C09128=1229.278,90.724,-47.007,-178.525,5.501,148.518
C09129=1229.283,90.475,-46.989,-178.527,5.501,148.519
C09130=1229.288,90.225,-46.971,-178.530,5.500,148.520
C09131=1229.292,89.976,-46.952,-178.532,5.499,148.520
C09132=1229.298,89.727,-46.933,-178.535,5.499,148.521
C09133=1229.303,89.478,-46.915,-178.537,5.498,148.521
C09134=1229.307,89.228,-46.898,-178.540,5.497,148.522
C09135=1229.312,88.979,-46.879,-178.542,5.496,148.522
C09136=1229.316,88.730,-46.860,-178.544,5.496,148.523
C09137=1229.321,88.481,-46.842,-178.548,5.494,148.524
C09138=1229.327,88.231,-46.824,-178.550,5.494,148.524
C09139=1229.331,87.981,-46.806,-178.552,5.493,148.525
C09140=1229.336,87.732,-46.788,-178.555,5.492,148.525
C09141=1229.341,87.483,-46.770,-178.558,5.492,148.526
C09142=1229.346,87.234,-46.752,-178.560,5.491,148.527
C09143=1229.351,86.985,-46.734,-178.562,5.490,148.527
C09144=1229.355,86.735,-46.715,-178.565,5.489,148.528
C09145=1229.360,86.486,-46.697,-178.568,5.489,148.528
C09146=1229.365,86.237,-46.678,-178.570,5.488,148.529
C09147=1229.370,85.988,-46.660,-178.572,5.487,148.529
C09148=1229.375,85.738,-46.642,-178.576,5.486,148.530
C09149=1229.380,85.489,-46.624,-178.578,5.485,148.531
C09150=1229.384,85.239,-46.606,-178.581,5.485,148.531
C09151=1229.389,84.990,-46.588,-178.583,5.484,148.532
C09152=1229.394,84.741,-46.570,-178.586,5.483,148.533
C09153=1229.399,84.492,-46.552,-178.588,5.482,148.533
C09154=1229.404,84.243,-46.534,-178.591,5.482,148.534
C09155=1229.408,83.993,-46.515,-178.593,5.481,148.534
C09156=1229.413,83.744,-46.497,-178.596,5.480,148.535
C09157=1229.418,83.494,-46.480,-178.598,5.480,148.536
C09158=1229.423,83.245,-46.462,-178.601,5.479,148.536
C09159=1229.428,82.996,-46.444,-178.604,5.479,148.537
C09160=1229.433,82.747,-46.426,-178.606,5.478,148.537
C09161=1229.438,82.498,-46.408,-178.609,5.476,148.538
C09162=1229.442,82.248,-46.389,-178.611,5.476,148.539
C09163=1229.448,81.979,-46.369,-178.614,5.475,148.539
C09164=1229.453,81.711,-46.350,-178.617,5.474,148.540
C09165=1229.459,81.443,-46.332,-178.619,5.474,148.541
C09166=1229.464,81.175,-46.312,-178.622,5.473,148.541
C09167=1229.468,80.925,-46.294,-178.625,5.472,148.542
C09168=1229.473,80.676,-46.276,-178.627,5.471,148.542
C09169=1229.478,80.426,-46.258,-178.630,5.470,148.543
C09170=1229.483,80.177,-46.240,-178.633,5.470,148.544
C09171=1229.488,79.928,-46.222,-178.635,5.469,148.544
C09172=1229.493,79.678,-46.205,-178.637,5.468,148.545
C09173=1229.498,79.429,-46.187,-178.640,5.467,148.545
C09174=1229.503,79.180,-46.169,-178.643,5.467,148.546
C09175=1229.508,78.931,-46.151,-178.645,5.466,148.547
C09176=1229.512,78.682,-46.133,-178.648,5.466,148.547
C09177=1229.517,78.433,-46.115,-178.650,5.465,148.548
C09178=1229.522,78.183,-46.098,-178.653,5.464,148.548
C09179=1229.527,77.933,-46.080,-178.655,5.464,148.549
C09180=1229.532,77.684,-46.062,-178.658,5.463,148.550
C09181=1229.537,77.435,-46.044,-178.660,5.462,148.550
C09182=1229.541,77.186,-46.026,-178.663,5.461,148.551
C09183=1229.547,76.936,-46.008,-178.665,5.461,148.551
C09184=1229.552,76.687,-45.990,-178.668,5.460,148.552
C09185=1229.556,76.438,-45.973,-178.670,5.460,148.553
C09186=1229.561,76.188,-45.955,-178.673,5.459,148.553
C09187=1229.566,75.939,-45.938,-178.676,5.457,148.554
C09188=1229.571,75.690,-45.920,-178.678,5.457,148.555
C09189=1229.576,75.440,-45.902,-178.681,5.456,148.555
C09190=1229.581,75.191,-45.885,-178.684,5.456,148.556
C09191=1229.586,74.941,-45.867,-178.686,5.455,148.556
C09192=1229.590,74.693,-45.849,-178.688,5.454,148.557
C09193=1229.595,74.443,-45.832,-178.691,5.453,148.558
C09194=1229.600,74.194,-45.814,-178.694,5.453,148.558
C09195=1229.605,73.944,-45.796,-178.696,5.452,148.559
C09196=1229.610,73.695,-45.779,-178.698,5.451,148.559
C09197=1229.614,73.446,-45.761,-178.701,5.451,148.560
C09198=1229.619,73.197,-45.743,-178.704,5.450,148.561
C09199=1229.625,72.947,-45.726,-178.706,5.449,148.561
C09200=1229.629,72.698,-45.708,-178.709,5.449,148.562
C09201=1229.634,72.448,-45.690,-178.711,5.448,148.562
C09202=1229.639,72.199,-45.674,-178.714,5.447,148.563
C09203=1229.644,71.950,-45.656,-178.716,5.447,148.564
C09204=1229.649,71.700,-45.638,-178.719,5.446,148.564
C09205=1229.654,71.451,-45.620,-178.722,5.446,148.565
C09206=1229.658,71.201,-45.604,-178.724,5.445,148.565
C09207=1229.663,70.952,-45.586,-178.726,5.444,148.566
C09208=1229.668,70.703,-45.568,-178.729,5.443,148.567
C09209=1229.673,70.453,-45.550,-178.732,5.443,148.567
C09210=1229.678,70.204,-45.533,-178.734,5.442,148.568
C09211=1229.683,69.954,-45.516,-178.737,5.442,148.569
C09212=1229.688,69.706,-45.498,-178.739,5.441,148.569
C09213=1229.693,69.457,-45.481,-178.742,5.440,148.570
C09214=1229.698,69.207,-45.463,-178.744,5.440,148.571
C09215=1229.703,68.958,-45.446,-178.747,5.439,148.571
C09216=1229.708,68.708,-45.428,-178.750,5.438,148.572
C09217=1229.712,68.459,-45.412,-178.752,5.438,148.572
C09218=1229.717,68.210,-45.394,-178.754,5.437,148.573
C09219=1229.722,67.960,-45.376,-178.757,5.436,148.574
C09220=1229.727,67.710,-45.360,-178.760,5.436,148.574
C09221=1229.732,67.461,-45.342,-178.762,5.435,148.575
C09222=1229.736,67.212,-45.325,-178.765,5.435,148.576
C09223=1229.741,66.963,-45.307,-178.767,5.434,148.576
C09224=1229.747,66.713,-45.290,-178.770,5.433,148.577
C09225=1229.751,66.465,-45.273,-178.772,5.432,148.577
C09226=1229.756,66.215,-45.255,-178.775,5.432,148.578
C09227=1229.762,65.965,-45.238,-178.777,5.431,148.579
C09228=1229.766,65.716,-45.221,-178.780,5.431,148.579
C09229=1229.771,65.466,-45.204,-178.782,5.430,148.580
C09230=1229.776,65.217,-45.187,-178.785,5.429,148.580
C09231=1229.780,64.968,-45.169,-178.788,5.429,148.581
C09232=1229.786,64.719,-45.152,-178.790,5.428,148.582
C09233=1229.791,64.469,-45.135,-178.793,5.427,148.582
C09234=1229.796,64.220,-45.117,-178.795,5.427,148.583
C09235=1229.800,63.970,-45.101,-178.798,5.426,148.584
C09236=1229.805,63.721,-45.083,-178.800,5.425,148.584
C09237=1229.810,63.471,-45.065,-178.803,5.425,148.585
C09238=1229.815,63.222,-45.049,-178.805,5.424,148.586
C09239=1229.821,62.973,-45.032,-178.808,5.424,148.586
C09240=1229.825,62.724,-45.015,-178.811,5.423,148.587
C09241=1229.830,62.474,-44.997,-178.813,5.422,148.588
C09242=1229.834,62.225,-44.981,-178.815,5.421,148.588
C09243=1229.840,61.975,-44.963,-178.818,5.421,148.589
C09244=1229.844,61.726,-44.946,-178.821,5.420,148.589
C09245=1229.850,61.477,-44.929,-178.823,5.420,148.590
C09246=1229.854,61.228,-44.912,-178.825,5.420,148.591
C09247=1229.859,60.978,-44.895,-178.828,5.419,148.591
C09248=1229.864,60.728,-44.878,-178.831,5.419,148.592
C09249=1229.869,60.479,-44.860,-178.833,5.418,148.592
C09250=1229.874,60.230,-44.844,-178.835,5.417,148.593
C09251=1229.879,59.981,-44.827,-178.838,5.417,148.594
C09252=1229.884,59.731,-44.810,-178.841,5.416,148.594
C09253=1229.889,59.481,-44.793,-178.843,5.416,148.595
C09254=1229.894,59.232,-44.777,-178.846,5.415,148.596
C09255=1229.899,58.983,-44.759,-178.849,5.414,148.596
C09256=1229.903,58.734,-44.742,-178.851,5.413,148.597
C09257=1229.908,58.484,-44.725,-178.853,5.413,148.597
C09258=1229.913,58.234,-44.708,-178.856,5.412,148.598
C09259=1229.918,57.986,-44.692,-178.859,5.412,148.599
C09260=1229.923,57.736,-44.674,-178.861,5.411,148.599
C09261=1229.928,57.486,-44.658,-178.864,5.411,148.600
C09262=1229.933,57.237,-44.641,-178.867,5.410,148.601
C09263=1229.938,56.988,-44.624,-178.869,5.409,148.601
C09264=1229.943,56.739,-44.606,-178.871,5.409,148.602
C09265=1229.947,56.489,-44.590,-178.874,5.408,148.603
C09266=1229.952,56.240,-44.573,-178.877,5.407,148.603
C09267=1229.958,55.972,-44.555,-178.879,5.407,148.604
C09268=1229.963,55.703,-44.538,-178.882,5.406,148.605
C09269=1229.969,55.434,-44.519,-178.885,5.406,148.605
C09270=1229.973,55.166,-44.501,-178.887,5.405,148.606
C09271=1229.979,54.917,-44.484,-178.890,5.404,148.607
C09272=1229.984,54.667,-44.467,-178.892,5.404,148.607
C09273=1229.988,54.418,-44.451,-178.895,5.403,148.608
C09274=1229.994,54.168,-44.434,-178.898,5.403,148.609
C09275=1229.999,53.919,-44.417,-178.900,5.402,148.609
C09276=1230.003,53.670,-44.400,-178.902,5.402,148.610
C09277=1230.008,53.421,-44.384,-178.905,5.402,148.611
C09278=1230.013,53.171,-44.367,-178.907,5.401,148.611
C09279=1230.018,52.921,-44.350,-178.910,5.400,148.612
C09280=1230.023,52.673,-44.334,-178.912,5.400,148.612
C09281=1230.028,52.423,-44.317,-178.915,5.399,148.613
C09282=1230.033,52.173,-44.300,-178.918,5.399,148.614
C09283=1230.037,51.924,-44.283,-178.920,5.398,148.614
C09284=1230.043,51.675,-44.266,-178.923,5.397,148.615
C09285=1230.047,51.425,-44.250,-178.926,5.397,148.616
C09286=1230.053,51.176,-44.234,-178.928,5.396,148.616
C09287=1230.057,50.926,-44.217,-178.930,5.395,148.617
C09288=1230.062,50.677,-44.200,-178.933,5.395,148.618
C09289=1230.068,50.428,-44.184,-178.935,5.395,148.618
C09290=1230.072,50.178,-44.167,-178.938,5.395,148.619
C09291=1230.076,49.929,-44.150,-178.940,5.394,148.620
C09292=1230.082,49.680,-44.134,-178.943,5.393,148.620
C09293=1230.087,49.430,-44.118,-178.946,5.393,148.621
C09294=1230.092,49.180,-44.101,-178.948,5.392,148.622
C09295=1230.097,48.931,-44.085,-178.951,5.392,148.622
C09296=1230.102,48.682,-44.067,-178.953,5.391,148.623
C09297=1230.107,48.433,-44.051,-178.956,5.390,148.623
C09298=1230.112,48.183,-44.035,-178.958,5.390,148.624
C09299=1230.116,47.933,-44.018,-178.961,5.389,148.625
C09300=1230.121,47.684,-44.002,-178.963,5.389,148.625
C09301=1230.127,47.435,-43.985,-178.966,5.389,148.626
C09302=1230.131,47.185,-43.968,-178.968,5.388,148.627
C09303=1230.136,46.936,-43.953,-178.971,5.388,148.627
C09304=1230.141,46.686,-43.936,-178.974,5.387,148.628
C09305=1230.146,46.438,-43.920,-178.976,5.386,148.629
C09306=1230.151,46.187,-43.904,-178.978,5.386,148.629
C09307=1230.157,45.938,-43.887,-178.981,5.385,148.630
C09308=1230.161,45.689,-43.870,-178.984,5.384,148.630
C09309=1230.166,45.439,-43.853,-178.986,5.384,148.631
C09310=1230.171,45.190,-43.838,-178.988,5.384,148.632
C09311=1230.175,44.940,-43.821,-178.991,5.384,148.632
C09312=1230.180,44.692,-43.805,-178.994,5.383,148.633
C09313=1230.185,44.442,-43.789,-178.996,5.382,148.634
C09314=1230.190,44.193,-43.773,-178.999,5.382,148.635
C09315=1230.196,43.943,-43.755,-179.002,5.381,148.635
C09316=1230.201,43.694,-43.740,-179.004,5.381,148.636
C09317=1230.205,43.444,-43.723,-179.006,5.380,148.636
C09318=1230.210,43.194,-43.707,-179.009,5.379,148.637
C09319=1230.215,42.945,-43.691,-179.011,5.379,148.638
C09320=1230.220,42.696,-43.674,-179.014,5.379,148.638
C09321=1230.225,42.446,-43.659,-179.016,5.378,148.639
C09322=1230.230,42.197,-43.642,-179.019,5.378,148.640
C09323=1230.235,41.947,-43.626,-179.022,5.377,148.640
C09324=1230.239,41.698,-43.610,-179.024,5.377,148.641
C09325=1230.245,41.449,-43.593,-179.027,5.376,148.642
C09326=1230.249,41.199,-43.577,-179.030,5.376,148.642
C09327=1230.254,40.950,-43.561,-179.032,5.376,148.643
C09328=1230.259,40.700,-43.545,-179.034,5.375,148.644
C09329=1230.264,40.451,-43.529,-179.036,5.374,148.644
C09330=1230.269,40.201,-43.513,-179.039,5.374,148.645
C09331=1230.275,39.952,-43.496,-179.042,5.373,148.646
C09332=1230.280,39.702,-43.480,-179.044,5.373,148.646
C09333=1230.285,39.453,-43.464,-179.047,5.372,148.647
C09334=1230.290,39.203,-43.448,-179.050,5.371,148.648
C09335=1230.295,38.954,-43.431,-179.052,5.372,148.648
C09336=1230.300,38.705,-43.416,-179.054,5.371,148.649
C09337=1230.305,38.456,-43.399,-179.057,5.371,148.650
C09338=1230.309,38.206,-43.384,-179.060,5.370,148.650
C09339=1230.314,37.957,-43.368,-179.062,5.369,148.651
C09340=1230.319,37.708,-43.352,-179.065,5.369,148.652
C09341=1230.324,37.457,-43.336,-179.068,5.368,148.652
C09342=1230.329,37.209,-43.320,-179.070,5.369,148.653
C09343=1230.334,36.959,-43.304,-179.072,5.368,148.653
C09344=1230.339,36.710,-43.287,-179.074,5.367,148.654
C09345=1230.344,36.460,-43.271,-179.077,5.367,148.655
C09346=1230.349,36.211,-43.255,-179.080,5.366,148.655
C09347=1230.354,35.962,-43.240,-179.082,5.365,148.656
C09348=1230.359,35.711,-43.224,-179.085,5.365,148.657
C09349=1230.364,35.463,-43.207,-179.087,5.365,148.657
C09350=1230.369,35.213,-43.191,-179.090,5.365,148.658
C09351=1230.374,34.963,-43.176,-179.092,5.364,148.659
C09352=1230.379,34.714,-43.160,-179.095,5.363,148.659
C09353=1230.383,34.465,-43.144,-179.098,5.363,148.660
C09354=1230.389,34.215,-43.129,-179.100,5.362,148.661
C09355=1230.393,33.966,-43.112,-179.102,5.363,148.662
C09356=1230.398,33.716,-43.096,-179.105,5.362,148.662
C09357=1230.404,33.467,-43.081,-179.108,5.362,148.663
C09358=1230.408,33.217,-43.064,-179.110,5.361,148.664
C09359=1230.414,32.968,-43.048,-179.112,5.360,148.664
C09360=1230.418,32.718,-43.033,-179.115,5.359,148.665
C09361=1230.423,32.469,-43.017,-179.118,5.359,148.665
C09362=1230.428,32.220,-43.001,-179.120,5.359,148.666
C09363=1230.433,31.970,-42.985,-179.122,5.359,148.667
C09364=1230.438,31.721,-42.970,-179.125,5.358,148.667
C09365=1230.443,31.472,-42.953,-179.128,5.358,148.668
C09366=1230.448,31.222,-42.937,-179.130,5.357,148.669
C09367=1230.453,30.973,-42.922,-179.133,5.356,148.669
C09368=1230.458,30.722,-42.906,-179.135,5.357,148.670
C09369=1230.463,30.473,-42.891,-179.138,5.356,148.671
C09370=1230.468,30.224,-42.875,-179.140,5.356,148.671
C09371=1230.474,29.956,-42.858,-179.143,5.355,148.672
C09372=1230.478,29.686,-42.841,-179.146,5.354,148.673
C09373=1230.484,29.418,-42.824,-179.148,5.354,148.673
C09374=1230.489,29.149,-42.807,-179.151,5.354,148.674
C09375=1230.495,28.900,-42.792,-179.154,5.353,148.675
C09376=1230.499,28.650,-42.775,-179.157,5.353,148.676
C09377=1230.504,28.401,-42.760,-179.158,5.353,148.676
C09378=1230.509,28.152,-42.745,-179.161,5.352,148.677
C09379=1230.514,27.902,-42.729,-179.164,5.351,148.678
C09380=1230.519,27.652,-42.713,-179.166,5.351,148.678
C09381=1230.524,27.403,-42.698,-179.169,5.350,148.679
C09382=1230.529,27.154,-42.682,-179.171,5.351,148.680
C09383=1230.534,26.904,-42.667,-179.174,5.350,148.680
C09384=1230.539,26.655,-42.652,-179.176,5.349,148.681
C09385=1230.544,26.406,-42.635,-179.179,5.349,148.682
C09386=1230.549,26.156,-42.619,-179.181,5.348,148.682
C09387=1230.554,25.906,-42.604,-179.184,5.348,148.683
C09388=1230.559,25.657,-42.589,-179.186,5.348,148.684
C09389=1230.564,25.408,-42.573,-179.189,5.348,148.684
C09390=1230.569,25.158,-42.557,-179.191,5.347,148.685
C09391=1230.574,24.909,-42.542,-179.194,5.346,148.686
C09392=1230.579,24.659,-42.527,-179.197,5.346,148.686
C09393=1230.584,24.410,-42.511,-179.199,5.346,148.687
C09394=1230.588,24.160,-42.496,-179.201,5.346,148.688
C09395=1230.594,23.911,-42.480,-179.204,5.345,148.688
C09396=1230.599,23.661,-42.464,-179.207,5.345,148.689
C09397=1230.604,23.412,-42.449,-179.209,5.344,148.690
C09398=1230.609,23.162,-42.434,-179.211,5.344,148.690
C09399=1230.613,22.913,-42.419,-179.214,5.344,148.691
C09400=1230.619,22.664,-42.403,-179.217,5.343,148.692
C09401=1230.624,22.414,-42.387,-179.219,5.343,148.693
C09402=1230.628,22.164,-42.372,-179.222,5.342,148.693
C09403=1230.634,21.915,-42.356,-179.224,5.342,148.694
C09404=1230.638,21.665,-42.342,-179.227,5.342,148.695
C09405=1230.644,21.416,-42.327,-179.229,5.341,148.695
C09406=1230.649,21.167,-42.311,-179.232,5.341,148.696
C09407=1230.653,20.917,-42.296,-179.234,5.340,148.696
C09408=1230.659,20.667,-42.280,-179.236,5.340,148.697
C09409=1230.663,20.418,-42.265,-179.239,5.339,148.698
C09410=1230.669,20.169,-42.249,-179.242,5.339,148.698
C09411=1230.674,19.919,-42.234,-179.244,5.338,148.699
C09412=1230.678,19.670,-42.218,-179.247,5.338,148.700
C09413=1230.684,19.420,-42.204,-179.249,5.338,148.700
C09414=1230.688,19.171,-42.189,-179.252,5.338,148.701
C09415=1230.694,18.921,-42.173,-179.254,5.337,148.702
C09416=1230.699,18.672,-42.158,-179.257,5.336,148.703
C09417=1230.703,18.422,-42.142,-179.259,5.337,148.703
C09418=1230.708,18.173,-42.127,-179.262,5.336,148.704
C09419=1230.714,17.923,-42.112,-179.264,5.336,148.705
C09420=1230.718,17.674,-42.097,-179.267,5.335,148.705
C09421=1230.724,17.424,-42.082,-179.270,5.335,148.706
C09422=1230.728,17.175,-42.067,-179.272,5.335,148.707
C09423=1230.733,16.925,-42.051,-179.274,5.334,148.707
C09424=1230.738,16.675,-42.036,-179.277,5.334,148.708
C09425=1230.743,16.426,-42.021,-179.280,5.333,148.709
C09426=1230.748,16.177,-42.006,-179.282,5.334,148.709
C09427=1230.753,15.928,-41.990,-179.284,5.333,148.710
C09428=1230.758,15.678,-41.976,-179.287,5.332,148.711
C09429=1230.764,15.428,-41.960,-179.290,5.332,148.711
C09430=1230.768,15.179,-41.945,-179.292,5.331,148.712
C09431=1230.773,14.929,-41.929,-179.294,5.332,148.713
C09432=1230.778,14.680,-41.915,-179.297,5.331,148.713
C09433=1230.784,14.430,-41.900,-179.300,5.331,148.714
C09434=1230.788,14.181,-41.885,-179.302,5.330,148.715
C09435=1230.793,13.931,-41.870,-179.304,5.330,148.716
C09436=1230.799,13.682,-41.855,-179.307,5.330,148.716
C09437=1230.803,13.433,-41.840,-179.310,5.329,148.717
C09438=1230.809,13.183,-41.825,-179.312,5.329,148.718
C09439=1230.814,12.934,-41.810,-179.314,5.329,148.718
C09440=1230.818,12.684,-41.794,-179.317,5.328,148.719
C09441=1230.823,12.434,-41.780,-179.320,5.328,148.720
C09442=1230.828,12.185,-41.765,-179.322,5.327,148.720
C09443=1230.834,11.935,-41.750,-179.324,5.328,148.721
C09444=1230.838,11.686,-41.735,-179.327,5.327,148.722
C09445=1230.843,11.437,-41.720,-179.330,5.327,148.722
C09446=1230.849,11.187,-41.705,-179.332,5.326,148.723
C09447=1230.853,10.938,-41.690,-179.334,5.326,148.724
C09448=1230.858,10.688,-41.676,-179.337,5.326,148.724
C09449=1230.864,10.438,-41.660,-179.340,5.325,148.725
C09450=1230.868,10.189,-41.645,-179.342,5.325,148.726
C09451=1230.873,9.940,-41.631,-179.344,5.325,148.726
C09452=1230.879,9.690,-41.615,-179.347,5.324,148.727
C09453=1230.884,9.440,-41.601,-179.350,5.324,148.728
C09454=1230.888,9.191,-41.586,-179.352,5.323,148.729
C09455=1230.894,8.941,-41.571,-179.354,5.324,148.729
C09456=1230.899,8.692,-41.556,-179.357,5.323,148.730
C09457=1230.904,8.443,-41.542,-179.360,5.323,148.731
C09458=1230.909,8.193,-41.526,-179.362,5.322,148.731
C09459=1230.914,7.943,-41.512,-179.365,5.322,148.732
C09460=1230.918,7.694,-41.497,-179.367,5.322,148.733
C09461=1230.924,7.444,-41.482,-179.370,5.321,148.733
C09462=1230.928,7.195,-41.467,-179.372,5.321,148.734
C09463=1230.933,6.945,-41.452,-179.375,5.321,148.735
C09464=1230.938,6.696,-41.437,-179.377,5.320,148.735
C09465=1230.944,6.446,-41.423,-179.380,5.320,148.736
C09466=1230.948,6.197,-41.408,-179.382,5.319,148.737
C09467=1230.953,5.947,-41.393,-179.385,5.320,148.737
C09468=1230.958,5.697,-41.379,-179.387,5.319,148.738
C09469=1230.964,5.448,-41.363,-179.390,5.319,148.739
C09470=1230.969,5.199,-41.349,-179.393,5.318,148.740
C09471=1230.974,4.950,-41.334,-179.395,5.318,148.740
C09472=1230.979,4.700,-41.320,-179.397,5.318,148.741
C09473=1230.984,4.450,-41.305,-179.400,5.317,148.742
C09474=1230.989,4.201,-41.290,-179.402,5.318,148.742
C09475=1230.994,3.932,-41.275,-179.405,5.317,148.743
C09476=1230.999,3.663,-41.259,-179.408,5.317,148.744
C09477=1231.005,3.394,-41.243,-179.410,5.316,148.745
C09478=1231.011,3.125,-41.228,-179.413,5.316,148.745
C09479=1231.015,2.876,-41.213,-179.416,5.315,148.746
C09480=1231.020,2.626,-41.198,-179.418,5.316,148.747
C09481=1231.025,2.376,-41.184,-179.420,5.315,148.747
C09482=1231.031,2.127,-41.169,-179.423,5.314,148.748
C09483=1231.035,1.877,-41.154,-179.426,5.314,148.749
C09484=1231.040,1.627,-41.140,-179.428,5.314,148.749
C09485=1231.045,1.378,-41.125,-179.431,5.314,148.750
C09486=1231.050,1.129,-41.111,-179.433,5.313,148.751
C09487=1231.056,0.880,-41.097,-179.435,5.313,148.751
C09488=1231.061,0.630,-41.082,-179.438,5.313,148.752
C09489=1231.066,0.381,-41.067,-179.441,5.312,148.753
C09490=1231.071,0.131,-41.053,-179.443,5.312,148.754
C09491=1231.076,-0.119,-41.038,-179.445,5.312,148.754
C09492=1231.081,-0.369,-41.024,-179.448,5.312,148.755
C09493=1231.085,-0.618,-41.009,-179.451,5.311,148.756
C09494=1231.090,-0.867,-40.995,-179.453,5.311,148.756
C09495=1231.095,-1.117,-40.981,-179.455,5.311,148.757
C09496=1231.100,-1.367,-40.966,-179.458,5.310,148.758
C09497=1231.106,-1.616,-40.952,-179.461,5.310,148.758
C09498=1231.111,-1.865,-40.937,-179.463,5.310,148.759
C09499=1231.116,-2.115,-40.922,-179.465,5.310,148.760
C09500=1231.121,-2.365,-40.908,-179.468,5.309,148.760
C09501=1231.126,-2.614,-40.894,-179.470,5.309,148.761
C09502=1231.131,-2.864,-40.880,-179.473,5.309,148.762
C09503=1231.136,-3.114,-40.865,-179.475,5.308,148.762
C09504=1231.141,-3.363,-40.850,-179.477,5.309,148.763
C09505=1231.146,-3.612,-40.836,-179.480,5.308,148.764
C09506=1231.151,-3.862,-40.822,-179.483,5.307,148.765
C09507=1231.156,-4.111,-40.808,-179.486,5.307,148.765
C09508=1231.161,-4.361,-40.794,-179.488,5.308,148.766
C09509=1231.166,-4.611,-40.779,-179.491,5.307,148.767
C09510=1231.171,-4.860,-40.765,-179.493,5.307,148.768
C09511=1231.177,-5.109,-40.751,-179.495,5.307,148.768
C09512=1231.182,-5.359,-40.737,-179.498,5.306,148.769
C09513=1231.186,-5.608,-40.722,-179.501,5.306,148.770
C09514=1231.191,-5.858,-40.708,-179.503,5.306,148.770
C09515=1231.196,-6.108,-40.693,-179.505,5.306,148.771
C09516=1231.201,-6.357,-40.679,-179.508,5.305,148.772
C09517=1231.207,-6.606,-40.665,-179.511,5.305,148.772
C09518=1231.212,-6.856,-40.651,-179.513,5.305,148.773
C09519=1231.216,-7.106,-40.637,-179.515,5.304,148.774
C09520=1231.221,-7.356,-40.622,-179.518,5.304,148.774
C09521=1231.226,-7.605,-40.608,-179.520,5.304,148.775
C09522=1231.232,-7.854,-40.594,-179.523,5.304,148.776
C09523=1231.237,-8.104,-40.580,-179.526,5.303,148.777
C09524=1231.242,-8.354,-40.566,-179.528,5.303,148.777
C09525=1231.247,-8.603,-40.551,-179.530,5.303,148.778
C09526=1231.252,-8.853,-40.537,-179.533,5.302,148.779
C09527=1231.257,-9.102,-40.524,-179.535,5.303,148.779
C09528=1231.262,-9.352,-40.509,-179.538,5.302,148.780
C09529=1231.266,-9.601,-40.495,-179.540,5.302,148.781
C09530=1231.271,-9.851,-40.481,-179.542,5.302,148.781
C09531=1231.277,-10.100,-40.467,-179.545,5.301,148.782
C09532=1231.282,-10.350,-40.453,-179.548,5.301,148.783
C09533=1231.287,-10.600,-40.439,-179.550,5.300,148.783
C09534=1231.292,-10.850,-40.425,-179.552,5.301,148.784
C09535=1231.298,-11.099,-40.411,-179.555,5.300,148.785
C09536=1231.303,-11.348,-40.397,-179.558,5.300,148.786
C09537=1231.307,-11.598,-40.383,-179.560,5.300,148.786
C09538=1231.312,-11.848,-40.369,-179.562,5.299,148.787
C09539=1231.317,-12.097,-40.355,-179.565,5.299,148.788
C09540=1231.322,-12.346,-40.341,-179.567,5.299,148.788
C09541=1231.327,-12.596,-40.326,-179.570,5.299,148.789
C09542=1231.333,-12.846,-40.313,-179.573,5.298,148.790
C09543=1231.337,-13.095,-40.299,-179.575,5.299,148.791
C09544=1231.342,-13.345,-40.285,-179.578,5.298,148.791
C09545=1231.347,-13.594,-40.271,-179.580,5.298,148.792
C09546=1231.353,-13.843,-40.257,-179.582,5.298,148.793
C09547=1231.358,-14.093,-40.243,-179.585,5.297,148.793
C09548=1231.363,-14.343,-40.229,-179.588,5.297,148.794
C09549=1231.368,-14.592,-40.216,-179.590,5.297,148.795
C09550=1231.373,-14.842,-40.201,-179.593,5.297,148.795
C09551=1231.378,-15.092,-40.187,-179.595,5.296,148.796
C09552=1231.383,-15.341,-40.173,-179.597,5.296,148.797
C09553=1231.389,-15.591,-40.160,-179.600,5.296,148.798
C09554=1231.393,-15.840,-40.146,-179.603,5.295,148.798
C09555=1231.398,-16.090,-40.132,-179.605,5.296,148.799
C09556=1231.403,-16.339,-40.118,-179.607,5.295,148.800
C09557=1231.409,-16.589,-40.104,-179.610,5.295,148.800
C09558=1231.413,-16.839,-40.091,-179.612,5.295,148.801
C09559=1231.418,-17.088,-40.077,-179.615,5.295,148.802
C09560=1231.423,-17.337,-40.062,-179.617,5.294,148.802
C09561=1231.429,-17.588,-40.049,-179.619,5.294,148.803
C09562=1231.433,-17.837,-40.036,-179.622,5.294,148.804
C09563=1231.438,-18.086,-40.021,-179.625,5.293,148.804
C09564=1231.444,-18.337,-40.008,-179.627,5.294,148.805
C09565=1231.449,-18.586,-39.994,-179.630,5.293,148.806
C09566=1231.453,-18.835,-39.980,-179.632,5.293,148.807
C09567=1231.459,-19.085,-39.967,-179.634,5.293,148.807
C09568=1231.464,-19.334,-39.953,-179.637,5.292,148.808
C09569=1231.468,-19.584,-39.939,-179.639,5.293,148.809
C09570=1231.474,-19.833,-39.926,-179.642,5.292,148.810
C09571=1231.479,-20.083,-39.911,-179.645,5.292,148.810
C09572=1231.484,-20.333,-39.897,-179.647,5.292,148.811
C09573=1231.489,-20.582,-39.885,-179.650,5.292,148.812
C09574=1231.494,-20.832,-39.870,-179.652,5.291,148.812
C09575=1231.500,-21.081,-39.857,-179.654,5.292,148.813
C09576=1231.504,-21.331,-39.843,-179.657,5.291,148.814
C09577=1231.509,-21.581,-39.829,-179.660,5.291,148.814
C09578=1231.515,-21.830,-39.816,-179.662,5.291,148.815
C09579=1231.520,-22.099,-39.802,-179.664,5.290,148.816
C09580=1231.525,-22.369,-39.787,-179.667,5.290,148.817
C09581=1231.531,-22.637,-39.772,-179.670,5.290,148.817
C09582=1231.537,-22.907,-39.757,-179.672,5.290,148.818
C09583=1231.541,-23.157,-39.744,-179.675,5.289,148.819
C09584=1231.547,-23.406,-39.730,-179.678,5.289,148.820
C09585=1231.552,-23.656,-39.717,-179.680,5.289,148.820
C09586=1231.557,-23.905,-39.703,-179.682,5.289,148.821
C09587=1231.562,-24.155,-39.690,-179.685,5.288,148.822
C09588=1231.566,-24.405,-39.676,-179.687,5.289,148.822
C09589=1231.572,-24.654,-39.663,-179.690,5.288,148.823
C09590=1231.577,-24.904,-39.649,-179.692,5.288,148.824
C09591=1231.582,-25.153,-39.636,-179.694,5.288,148.824
C09592=1231.587,-25.403,-39.622,-179.697,5.287,148.825
C09593=1231.592,-25.652,-39.609,-179.699,5.288,148.826
C09594=1231.597,-25.902,-39.595,-179.702,5.287,148.827
C09595=1231.603,-26.151,-39.582,-179.705,5.287,148.827
C09596=1231.607,-26.401,-39.568,-179.707,5.287,148.828
C09597=1231.612,-26.651,-39.555,-179.710,5.287,148.829
C09598=1231.618,-26.901,-39.542,-179.712,5.287,148.830
C09599=1231.622,-27.150,-39.528,-179.715,5.287,148.830
C09600=1231.628,-27.400,-39.515,-179.717,5.286,148.831
C09601=1231.633,-27.649,-39.501,-179.719,5.286,148.832
C09602=1231.638,-27.899,-39.488,-179.722,5.286,148.832
C09603=1231.643,-28.149,-39.474,-179.725,5.285,148.833
C09604=1231.648,-28.398,-39.461,-179.727,5.286,148.834
C09605=1231.653,-28.648,-39.447,-179.729,5.285,148.834
C09606=1231.658,-28.897,-39.434,-179.731,5.286,148.835
C09607=1231.663,-29.147,-39.421,-179.734,5.285,148.836
C09608=1231.669,-29.396,-39.408,-179.737,5.285,148.837
C09609=1231.674,-29.646,-39.394,-179.739,5.285,148.837
C09610=1231.679,-29.895,-39.381,-179.741,5.284,148.838
C09611=1231.684,-30.146,-39.368,-179.744,5.284,148.839
C09612=1231.689,-30.394,-39.354,-179.746,5.284,148.839
C09613=1231.693,-30.644,-39.341,-179.749,5.284,148.840
C09614=1231.699,-30.894,-39.328,-179.751,5.284,148.841
C09615=1231.704,-31.143,-39.315,-179.754,5.283,148.841
C09616=1231.709,-31.393,-39.301,-179.756,5.283,148.842
C09617=1231.714,-31.642,-39.289,-179.758,5.283,148.843
C09618=1231.720,-31.893,-39.275,-179.762,5.283,148.844
C09619=1231.724,-32.141,-39.262,-179.764,5.283,148.844
C09620=1231.730,-32.392,-39.248,-179.766,5.283,148.845
C09621=1231.735,-32.641,-39.236,-179.769,5.282,148.846
C09622=1231.739,-32.891,-39.222,-179.771,5.283,148.847
C09623=1231.745,-33.140,-39.209,-179.774,5.282,148.847
C09624=1231.749,-33.390,-39.196,-179.776,5.282,148.848
C09625=1231.755,-33.640,-39.183,-179.778,5.282,148.849
C09626=1231.760,-33.889,-39.170,-179.781,5.282,148.849
C09627=1231.765,-34.139,-39.156,-179.783,5.282,148.850
C09628=1231.770,-34.388,-39.143,-179.786,5.281,148.851
C09629=1231.775,-34.638,-39.130,-179.788,5.281,148.851
C09630=1231.781,-34.888,-39.117,-179.791,5.281,148.852
C09631=1231.786,-35.137,-39.104,-179.793,5.281,148.853
C09632=1231.790,-35.387,-39.091,-179.795,5.281,148.854
C09633=1231.796,-35.636,-39.077,-179.798,5.280,148.854
C09634=1231.801,-35.886,-39.064,-179.801,5.280,148.855
C09635=1231.806,-36.135,-39.052,-179.803,5.280,148.856
C09636=1231.812,-36.385,-39.039,-179.805,5.280,148.856
C09637=1231.816,-36.635,-39.026,-179.807,5.280,148.857
C09638=1231.821,-36.884,-39.012,-179.810,5.280,148.858
C09639=1231.826,-37.134,-38.999,-179.813,5.279,148.859
C09640=1231.831,-37.383,-38.986,-179.815,5.280,148.859
C09641=1231.836,-37.633,-38.974,-179.818,5.279,148.860
C09642=1231.842,-37.883,-38.960,-179.820,5.280,148.861
C09643=1231.847,-38.132,-38.947,-179.823,5.279,148.861
C09644=1231.852,-38.382,-38.935,-179.825,5.279,148.862
C09645=1231.857,-38.632,-38.921,-179.828,5.279,148.863
C09646=1231.862,-38.881,-38.909,-179.830,5.278,148.864
C09647=1231.867,-39.131,-38.896,-179.832,5.279,148.864
C09648=1231.872,-39.380,-38.882,-179.835,5.278,148.865
C09649=1231.877,-39.630,-38.869,-179.838,5.278,148.866
C09650=1231.882,-39.880,-38.856,-179.840,5.278,148.866
C09651=1231.887,-40.129,-38.844,-179.842,5.278,148.867
C09652=1231.893,-40.379,-38.830,-179.844,5.278,148.868
C09653=1231.897,-40.629,-38.817,-179.847,5.277,148.868
C09654=1231.903,-40.878,-38.805,-179.850,5.277,148.869
C09655=1231.908,-41.127,-38.792,-179.852,5.277,148.870
C09656=1231.913,-41.378,-38.779,-179.855,5.277,148.871
C09657=1231.918,-41.627,-38.766,-179.857,5.277,148.871
C09658=1231.923,-41.876,-38.754,-179.859,5.277,148.872
C09659=1231.928,-42.126,-38.741,-179.861,5.277,148.873
C09660=1231.933,-42.376,-38.728,-179.864,5.276,148.873
C09661=1231.939,-42.625,-38.715,-179.867,5.276,148.874
C09662=1231.944,-42.875,-38.702,-179.869,5.277,148.875
C09663=1231.948,-43.125,-38.689,-179.872,5.276,148.876
C09664=1231.954,-43.374,-38.677,-179.874,5.276,148.876
C09665=1231.959,-43.623,-38.664,-179.877,5.276,148.877
C09666=1231.964,-43.874,-38.651,-179.879,5.275,148.878
C09667=1231.969,-44.124,-38.639,-179.881,5.276,148.878
C09668=1231.974,-44.373,-38.626,-179.884,5.275,148.879
C09669=1231.980,-44.622,-38.613,-179.886,5.276,148.880
C09670=1231.984,-44.872,-38.600,-179.889,5.275,148.881
C09671=1231.989,-45.122,-38.588,-179.891,5.275,148.881
C09672=1231.995,-45.371,-38.575,-179.894,5.275,148.882
C09673=1232.000,-45.621,-38.562,-179.896,5.274,148.883
C09674=1232.005,-45.870,-38.549,-179.898,5.275,148.883
C09675=1232.010,-46.120,-38.536,-179.901,5.274,148.884
C09676=1232.015,-46.370,-38.525,-179.903,5.275,148.885
C09677=1232.020,-46.620,-38.512,-179.906,5.274,148.886
C09678=1232.025,-46.869,-38.499,-179.908,5.274,148.886
C09679=1232.031,-47.119,-38.486,-179.910,5.274,148.887
C09680=1232.036,-47.368,-38.473,-179.913,5.273,148.888
C09681=1232.040,-47.618,-38.460,-179.915,5.274,148.888
C09682=1232.046,-47.868,-38.448,-179.918,5.273,148.889
C09683=1232.051,-48.137,-38.435,-179.920,5.274,148.890
C09684=1232.057,-48.407,-38.421,-179.923,5.273,148.891
C09685=1232.062,-48.677,-38.407,-179.926,5.273,148.891
C09686=1232.068,-48.946,-38.394,-179.929,5.273,148.892
C09687=1232.073,-49.196,-38.381,-179.931,5.273,148.893
C09688=1232.078,-49.446,-38.369,-179.934,5.273,148.894
C09689=1232.084,-49.695,-38.356,-179.936,5.273,148.894
C09690=1232.089,-49.945,-38.343,-179.939,5.273,148.895
C09691=1232.094,-50.195,-38.331,-179.941,5.273,148.896
C09692=1232.099,-50.445,-38.318,-179.943,5.272,148.897
C09693=1232.104,-50.694,-38.306,-179.946,5.272,148.897
C09694=1232.109,-50.943,-38.293,-179.948,5.272,148.898
C09695=1232.114,-51.193,-38.281,-179.951,5.272,148.899
C09696=1232.120,-51.443,-38.269,-179.953,5.272,148.899
C09697=1232.124,-51.693,-38.256,-179.955,5.272,148.900
C09698=1232.129,-51.942,-38.244,-179.958,5.272,148.901
C09699=1232.135,-52.192,-38.231,-179.960,5.271,148.901
C09700=1232.140,-52.441,-38.218,-179.962,5.272,148.902
C09701=1232.145,-52.691,-38.207,-179.965,5.271,148.903
C09702=1232.150,-52.941,-38.194,-179.968,5.271,148.904
C09703=1232.155,-53.190,-38.181,-179.970,5.271,148.904
C09704=1232.160,-53.440,-38.169,-179.972,5.271,148.905
C09705=1232.165,-53.690,-38.157,-179.974,5.271,148.906
C09706=1232.170,-53.939,-38.144,-179.977,5.270,148.906
C09707=1232.176,-54.189,-38.132,-179.980,5.271,148.907
C09708=1232.180,-54.439,-38.119,-179.982,5.271,148.908
C09709=1232.186,-54.688,-38.106,-179.984,5.271,148.909
C09710=1232.191,-54.938,-38.095,-179.987,5.271,148.909
C09711=1232.196,-55.187,-38.082,-179.990,5.270,148.910
C09712=1232.202,-55.437,-38.070,-179.992,5.270,148.911
C09713=1232.206,-55.686,-38.058,-179.995,5.270,148.912
C09714=1232.211,-55.936,-38.045,-179.997,5.270,148.912
C09715=1232.216,-56.186,-38.034,-179.999,5.270,148.913
C09716=1232.221,-56.436,-38.021,179.999,5.270,148.914
C09717=1232.226,-56.686,-38.009,179.996,5.270,148.914
C09718=1232.232,-56.935,-37.996,179.994,5.270,148.915
C09719=1232.237,-57.185,-37.984,179.991,5.269,148.916
C09720=1232.242,-57.434,-37.972,179.989,5.269,148.916
C09721=1232.247,-57.684,-37.959,179.986,5.269,148.917
C09722=1232.253,-57.933,-37.947,179.984,5.269,148.918
C09723=1232.258,-58.183,-37.935,179.982,5.269,148.919
C09724=1232.262,-58.432,-37.923,179.979,5.269,148.919
C09725=1232.267,-58.682,-37.910,179.977,5.269,148.920
C09726=1232.272,-58.932,-37.898,179.974,5.269,148.921
C09727=1232.278,-59.182,-37.886,179.972,5.269,148.921
C09728=1232.283,-59.432,-37.874,179.970,5.268,148.922
C09729=1232.288,-59.681,-37.861,179.967,5.269,148.923
C09730=1232.294,-59.931,-37.849,179.965,5.268,148.924
C09731=1232.298,-60.181,-37.838,179.962,5.268,148.924
C09732=1232.303,-60.430,-37.826,179.960,5.268,148.925
C09733=1232.309,-60.680,-37.814,179.957,5.268,148.926
C09734=1232.314,-60.929,-37.801,179.955,5.268,148.927
C09735=1232.319,-61.179,-37.789,179.952,5.268,148.927
C09736=1232.324,-61.428,-37.777,179.950,5.268,148.928
C09737=1232.329,-61.678,-37.765,179.947,5.268,148.929
C09738=1232.334,-61.927,-37.753,179.945,5.268,148.929
C09739=1232.340,-62.177,-37.741,179.943,5.268,148.930
C09740=1232.345,-62.428,-37.729,179.940,5.268,148.931
C09741=1232.350,-62.677,-37.716,179.938,5.267,148.932
C09742=1232.354,-62.927,-37.705,179.936,5.268,148.932
C09743=1232.360,-63.177,-37.693,179.933,5.267,148.933
C09744=1232.365,-63.426,-37.680,179.930,5.267,148.934
C09745=1232.370,-63.676,-37.668,179.928,5.267,148.934
C09746=1232.375,-63.925,-37.656,179.926,5.267,148.935
C09747=1232.380,-64.175,-37.644,179.924,5.267,148.936
C09748=1232.386,-64.425,-37.633,179.921,5.266,148.936
C09749=1232.391,-64.674,-37.620,179.919,5.267,148.937
C09750=1232.396,-64.924,-37.608,179.916,5.266,148.938
C09751=1232.401,-65.174,-37.597,179.914,5.267,148.939
C09752=1232.406,-65.423,-37.584,179.911,5.266,148.939
C09753=1232.411,-65.673,-37.572,179.909,5.267,148.940
C09754=1232.417,-65.923,-37.560,179.907,5.266,148.941
C09755=1232.421,-66.173,-37.549,179.905,5.266,148.941
C09756=1232.427,-66.422,-37.537,179.902,5.266,148.942
C09757=1232.432,-66.672,-37.525,179.900,5.266,148.943
C09758=1232.437,-66.921,-37.513,179.897,5.266,148.944
C09759=1232.442,-67.171,-37.501,179.894,5.265,148.944
C09760=1232.447,-67.421,-37.489,179.892,5.266,148.945
C09761=1232.453,-67.671,-37.477,179.890,5.265,148.946
C09762=1232.458,-67.920,-37.466,179.888,5.266,148.946
C09763=1232.463,-68.169,-37.453,179.885,5.265,148.947
C09764=1232.469,-68.419,-37.442,179.883,5.265,148.948
C09765=1232.473,-68.668,-37.430,179.880,5.265,148.948
C09766=1232.479,-68.918,-37.418,179.878,5.266,148.949
C09767=1232.484,-69.168,-37.406,179.875,5.265,148.950
C09768=1232.489,-69.417,-37.394,179.873,5.265,148.951
C09769=1232.494,-69.667,-37.383,179.870,5.265,148.952
C09770=1232.499,-69.917,-37.371,179.868,5.265,148.952
C09771=1232.504,-70.167,-37.359,179.865,5.265,148.953
C09772=1232.509,-70.417,-37.348,179.863,5.265,148.954
C09773=1232.515,-70.666,-37.335,179.861,5.265,148.954
C09774=1232.519,-70.916,-37.324,179.859,5.265,148.955
C09775=1232.525,-71.166,-37.312,179.856,5.265,148.956
C09776=1232.529,-71.415,-37.300,179.854,5.265,148.956
C09777=1232.535,-71.664,-37.289,179.851,5.265,148.957
C09778=1232.541,-71.914,-37.277,179.849,5.265,148.958
C09779=1232.546,-72.164,-37.266,179.846,5.264,148.959
C09780=1232.551,-72.414,-37.254,179.844,5.265,148.959
C09781=1232.556,-72.663,-37.241,179.842,5.264,148.960
C09782=1232.561,-72.913,-37.230,179.839,5.265,148.961
C09783=1232.566,-73.163,-37.218,179.837,5.264,148.961
C09784=1232.571,-73.412,-37.207,179.834,5.264,148.962
C09785=1232.576,-73.662,-37.195,179.832,5.264,148.963
C09786=1232.582,-73.912,-37.183,179.829,5.264,148.964
C09787=1232.587,-74.182,-37.171,179.827,5.264,148.964
C09788=1232.593,-74.453,-37.159,179.825,5.263,148.965
C09789=1232.598,-74.722,-37.146,179.822,5.264,148.966
C09790=1232.604,-74.993,-37.133,179.819,5.264,148.967
C09791=1232.609,-75.243,-37.121,179.817,5.263,148.967
C09792=1232.614,-75.492,-37.110,179.815,5.264,148.968
C09793=1232.619,-75.742,-37.098,179.812,5.263,148.969
C09794=1232.625,-75.991,-37.087,179.810,5.263,148.969
C09795=1232.630,-76.241,-37.075,179.807,5.263,148.970
C09796=1232.636,-76.491,-37.063,179.805,5.263,148.971
C09797=1232.640,-76.741,-37.052,179.802,5.263,148.972
C09798=1232.646,-76.991,-37.040,179.800,5.263,148.972
C09799=1232.650,-77.240,-37.029,179.798,5.263,148.973
C09800=1232.656,-77.489,-37.017,179.796,5.263,148.974
C09801=1232.661,-77.739,-37.006,179.793,5.263,148.974
C09802=1232.666,-77.989,-36.994,179.791,5.263,148.975
C09803=1232.671,-78.239,-36.983,179.788,5.262,148.976
C09804=1232.677,-78.489,-36.971,179.786,5.263,148.977
C09805=1232.681,-78.738,-36.960,179.783,5.262,148.977
C09806=1232.688,-78.988,-36.949,179.781,5.263,148.978
C09807=1232.692,-79.238,-36.938,179.779,5.262,148.979
C09808=1232.697,-79.487,-36.926,179.777,5.263,148.979
C09809=1232.702,-79.737,-36.915,179.774,5.262,148.980
C09810=1232.707,-79.987,-36.903,179.772,5.262,148.981
C09811=1232.713,-80.236,-36.892,179.769,5.262,148.982
C09812=1232.718,-80.486,-36.880,179.767,5.262,148.982
C09813=1232.723,-80.736,-36.869,179.764,5.262,148.983
C09814=1232.728,-80.985,-36.857,179.762,5.262,148.984
C09815=1232.733,-81.235,-36.845,179.760,5.262,148.984
C09816=1232.739,-81.485,-36.835,179.757,5.262,148.985
C09817=1232.744,-81.734,-36.824,179.755,5.262,148.986
C09818=1232.749,-81.984,-36.812,179.753,5.262,148.986
C09819=1232.754,-82.234,-36.801,179.750,5.262,148.987
C09820=1232.760,-82.483,-36.789,179.748,5.262,148.988
C09821=1232.765,-82.733,-36.778,179.745,5.261,148.989
C09822=1232.770,-82.983,-36.767,179.743,5.262,148.989
C09823=1232.775,-83.233,-36.755,179.740,5.261,148.990
C09824=1232.780,-83.483,-36.744,179.738,5.262,148.991
C09825=1232.785,-83.732,-36.733,179.736,5.261,148.991
C09826=1232.790,-83.981,-36.721,179.734,5.262,148.992
C09827=1232.795,-84.232,-36.711,179.731,5.261,148.993
C09828=1232.801,-84.482,-36.699,179.729,5.261,148.994
C09829=1232.806,-84.731,-36.688,179.726,5.261,148.994
C09830=1232.811,-84.980,-36.677,179.724,5.261,148.995
C09831=1232.816,-85.230,-36.665,179.721,5.261,148.996
C09832=1232.821,-85.480,-36.654,179.719,5.261,148.996
C09833=1232.827,-85.729,-36.643,179.717,5.261,148.997
C09834=1232.832,-85.979,-36.631,179.715,5.261,148.998
C09835=1232.837,-86.229,-36.620,179.712,5.261,148.999
C09836=1232.842,-86.478,-36.610,179.710,5.261,148.999
C09837=1232.848,-86.728,-36.598,179.707,5.261,149.000
C09838=1232.852,-86.978,-36.587,179.705,5.261,149.001
C09839=1232.857,-87.228,-36.576,179.702,5.260,149.001
C09840=1232.863,-87.477,-36.565,179.700,5.261,149.002
C09841=1232.868,-87.727,-36.553,179.698,5.260,149.003
C09842=1232.873,-87.977,-36.543,179.696,5.261,149.004
C09843=1232.878,-88.226,-36.532,179.693,5.260,149.004
C09844=1232.884,-88.476,-36.520,179.691,5.261,149.005
C09845=1232.889,-88.726,-36.509,179.688,5.260,149.006
C09846=1232.894,-88.975,-36.498,179.686,5.260,149.006
C09847=1232.899,-89.225,-36.487,179.683,5.260,149.007
C09848=1232.905,-89.476,-36.476,179.681,5.260,149.008
C09849=1232.910,-89.724,-36.465,179.679,5.261,149.009
C09850=1232.914,-89.974,-36.454,179.676,5.260,149.009
C09851=1232.919,-90.224,-36.443,179.674,5.261,149.010
C09852=1232.926,-90.474,-36.432,179.672,5.260,149.011
C09853=1232.930,-90.723,-36.420,179.670,5.261,149.011
C09854=1232.935,-90.973,-36.410,179.667,5.260,149.012
C09855=1232.940,-91.222,-36.399,179.665,5.260,149.013
C09856=1232.946,-91.473,-36.388,179.662,5.260,149.013
C09857=1232.951,-91.723,-36.376,179.660,5.260,149.014
C09858=1232.957,-91.972,-36.366,179.657,5.260,149.015
C09859=1232.961,-92.222,-36.355,179.655,5.260,149.016
C09860=1232.966,-92.471,-36.344,179.653,5.260,149.016
C09861=1232.972,-92.721,-36.333,179.651,5.260,149.017
C09862=1232.977,-92.971,-36.322,179.648,5.260,149.018
C09863=1232.983,-93.220,-36.311,179.646,5.260,149.018
C09864=1232.987,-93.470,-36.300,179.643,5.260,149.019
C09865=1232.992,-93.720,-36.290,179.641,5.260,149.020
C09866=1232.998,-93.969,-36.278,179.638,5.260,149.021
C09867=1233.003,-94.220,-36.267,179.636,5.260,149.021
C09868=1233.008,-94.469,-36.256,179.634,5.259,149.022
C09869=1233.014,-94.719,-36.246,179.631,5.260,149.023
C09870=1233.018,-94.968,-36.235,179.629,5.259,149.023
C09871=1233.024,-95.218,-36.224,179.627,5.260,149.024
C09872=1233.029,-95.468,-36.213,179.624,5.259,149.025
C09873=1233.034,-95.718,-36.202,179.622,5.260,149.026
C09874=1233.040,-95.967,-36.191,179.620,5.260,149.026
C09875=1233.045,-96.217,-36.180,179.617,5.259,149.027
C09876=1233.050,-96.466,-36.170,179.615,5.260,149.028
C09877=1233.055,-96.717,-36.159,179.612,5.259,149.028
C09878=1233.060,-96.966,-36.149,179.610,5.260,149.029
C09879=1233.065,-97.216,-36.137,179.608,5.259,149.030
C09880=1233.070,-97.466,-36.127,179.606,5.259,149.030
C09881=1233.076,-97.715,-36.115,179.603,5.259,149.031
C09882=1233.081,-97.965,-36.105,179.601,5.259,149.032
C09883=1233.086,-98.214,-36.094,179.599,5.259,149.032
C09884=1233.091,-98.465,-36.083,179.596,5.259,149.033
C09885=1233.097,-98.714,-36.073,179.594,5.259,149.034
C09886=1233.102,-98.964,-36.062,179.592,5.259,149.035
C09887=1233.107,-99.213,-36.052,179.589,5.259,149.035
C09888=1233.112,-99.464,-36.041,179.587,5.259,149.036
C09889=1233.117,-99.713,-36.030,179.584,5.258,149.037
C09890=1233.123,-99.963,-36.020,179.582,5.259,149.037
C09891=1233.128,-100.234,-36.007,179.579,5.258,149.038
C09892=1233.134,-100.504,-35.997,179.577,5.259,149.039
C09893=1233.140,-100.775,-35.984,179.574,5.259,149.040
C09894=1233.146,-101.047,-35.973,179.572,5.259,149.041
C09895=1233.151,-101.296,-35.962,179.569,5.259,149.041
C09896=1233.156,-101.546,-35.951,179.567,5.259,149.042
C09897=1233.161,-101.796,-35.941,179.565,5.259,149.043
C09898=1233.166,-102.045,-35.930,179.563,5.259,149.043
C09899=1233.172,-102.295,-35.920,179.560,5.258,149.044
C09900=1233.177,-102.545,-35.909,179.558,5.259,149.045
C09901=1233.182,-102.794,-35.898,179.555,5.258,149.046
C09902=1233.187,-103.044,-35.888,179.553,5.259,149.046
C09903=1233.193,-103.294,-35.877,179.550,5.258,149.047
C09904=1233.198,-103.544,-35.867,179.548,5.259,149.048
C09905=1233.203,-103.793,-35.856,179.546,5.258,149.048
C09906=1233.208,-104.043,-35.845,179.544,5.258,149.049
C09907=1233.213,-104.292,-35.836,179.542,5.259,149.050
C09908=1233.218,-104.543,-35.825,179.539,5.258,149.050
C09909=1233.223,-104.792,-35.814,179.537,5.258,149.051
C09910=1233.228,-105.042,-35.804,179.534,5.258,149.052
C09911=1233.234,-105.291,-35.793,179.532,5.258,149.052
C09912=1233.239,-105.542,-35.783,179.530,5.258,149.053
C09913=1233.244,-105.791,-35.773,179.528,5.258,149.054
C09914=1233.249,-106.041,-35.761,179.525,5.258,149.055
C09915=1233.255,-106.290,-35.751,179.523,5.258,149.055
C09916=1233.260,-106.541,-35.741,179.520,5.258,149.056
C09917=1233.265,-106.790,-35.730,179.518,5.258,149.057
C09918=1233.271,-107.040,-35.720,179.515,5.258,149.057
C09919=1233.276,-107.290,-35.710,179.513,5.258,149.058
C09920=1233.281,-107.539,-35.699,179.511,5.258,149.059
C09921=1233.286,-107.789,-35.688,179.509,5.258,149.060
C09922=1233.291,-108.038,-35.678,179.506,5.258,149.060
C09923=1233.296,-108.289,-35.668,179.504,5.258,149.061
C09924=1233.301,-108.538,-35.658,179.502,5.258,149.062
C09925=1233.307,-108.788,-35.648,179.499,5.257,149.062
C09926=1233.312,-109.038,-35.637,179.497,5.258,149.063
C09927=1233.318,-109.287,-35.627,179.495,5.257,149.064
C09928=1233.322,-109.537,-35.615,179.493,5.258,149.064
C09929=1233.328,-109.787,-35.605,179.490,5.257,149.065
C09930=1233.332,-110.036,-35.595,179.488,5.258,149.066
C09931=1233.338,-110.286,-35.585,179.485,5.257,149.067
C09932=1233.343,-110.536,-35.575,179.483,5.258,149.067
C09933=1233.348,-110.786,-35.564,179.481,5.258,149.068
C09934=1233.354,-111.035,-35.554,179.478,5.258,149.069
C09935=1233.360,-111.285,-35.544,179.476,5.258,149.069
C09936=1233.364,-111.535,-35.534,179.474,5.257,149.070
C09937=1233.369,-111.784,-35.524,179.471,5.258,149.071
C09938=1233.374,-112.035,-35.513,179.469,5.257,149.071
C09939=1233.380,-112.284,-35.503,179.467,5.257,149.072
C09940=1233.386,-112.534,-35.493,179.464,5.257,149.073
C09941=1233.391,-112.784,-35.482,179.462,5.257,149.073
C09942=1233.396,-113.033,-35.472,179.460,5.257,149.074
C09943=1233.401,-113.283,-35.462,179.458,5.257,149.075
C09944=1233.406,-113.533,-35.452,179.456,5.258,149.076
C09945=1233.412,-113.783,-35.441,179.453,5.257,149.076
C09946=1233.417,-114.033,-35.431,179.451,5.258,149.077
C09947=1233.422,-114.282,-35.421,179.448,5.257,149.078
C09948=1233.427,-114.532,-35.411,179.446,5.258,149.078
C09949=1233.432,-114.782,-35.401,179.443,5.257,149.079
C09950=1233.438,-115.031,-35.390,179.441,5.257,149.080
C09951=1233.443,-115.281,-35.381,179.439,5.257,149.080
C09952=1233.448,-115.531,-35.370,179.437,5.257,149.081
C09953=1233.453,-115.780,-35.360,179.434,5.257,149.082
C09954=1233.459,-116.030,-35.350,179.432,5.257,149.083
C09955=1233.463,-116.280,-35.340,179.430,5.257,149.083
C09956=1233.469,-116.530,-35.330,179.427,5.257,149.084
C09957=1233.475,-116.780,-35.320,179.425,5.257,149.085
C09958=1233.480,-117.029,-35.310,179.423,5.257,149.085
C09959=1233.484,-117.279,-35.300,179.420,5.257,149.086
C09960=1233.490,-117.529,-35.290,179.418,5.257,149.087
C09961=1233.496,-117.778,-35.279,179.416,5.257,149.088
C09962=1233.500,-118.028,-35.269,179.414,5.256,149.088
C09963=1233.506,-118.278,-35.259,179.411,5.257,149.089
C09964=1233.511,-118.528,-35.250,179.409,5.257,149.089
C09965=1233.516,-118.778,-35.240,179.407,5.257,149.090
C09966=1233.521,-119.027,-35.230,179.405,5.257,149.091
C09967=1233.527,-119.277,-35.219,179.402,5.257,149.092
C09968=1233.532,-119.526,-35.210,179.400,5.257,149.092
C09969=1233.537,-119.776,-35.199,179.397,5.257,149.093
C09970=1233.543,-120.026,-35.190,179.395,5.257,149.094
C09971=1233.547,-120.276,-35.180,179.392,5.256,149.094
C09972=1233.552,-120.526,-35.169,179.391,5.256,149.095
C09973=1233.558,-120.775,-35.159,179.389,5.257,149.096
C09974=1233.563,-121.025,-35.150,179.386,5.256,149.096
C09975=1233.569,-121.275,-35.140,179.384,5.257,149.097
C09976=1233.574,-121.525,-35.130,179.381,5.256,149.098
C09977=1233.579,-121.774,-35.120,179.379,5.257,149.099
C09978=1233.584,-122.024,-35.110,179.376,5.256,149.099
C09979=1233.590,-122.273,-35.100,179.374,5.257,149.100
C09980=1233.594,-122.524,-35.090,179.372,5.256,149.101
C09981=1233.600,-122.773,-35.080,179.370,5.256,149.101
C09982=1233.605,-123.023,-35.070,179.368,5.257,149.102
C09983=1233.611,-123.273,-35.061,179.365,5.256,149.103
C09984=1233.616,-123.523,-35.050,179.363,5.257,149.103
C09985=1233.621,-123.772,-35.041,179.360,5.256,149.104
C09986=1233.626,-124.022,-35.031,179.358,5.256,149.105
C09987=1233.631,-124.272,-35.022,179.356,5.256,149.106
C09988=1233.637,-124.521,-35.011,179.354,5.256,149.106
C09989=1233.641,-124.771,-35.001,179.351,5.256,149.107
C09990=1233.647,-125.021,-34.992,179.349,5.256,149.107
C09991=1233.653,-125.271,-34.982,179.347,5.256,149.108
C09992=1233.658,-125.520,-34.972,179.345,5.256,149.109
C09993=1233.664,-125.770,-34.963,179.342,5.256,149.110
C09994=1233.668,-126.020,-34.953,179.340,5.256,149.110
C09995=1233.247,-126.031,-34.988,179.335,5.259,149.112
C09996=1233.241,-125.781,-34.998,179.338,5.260,149.112
//INST
///DATE 2021/06/25 14:26
///ATTR SC,RW,RJ
////FRAME ROBOT
///GROUP1 RB1
NOP
MOVL C00000 V=800.0 PL=0
MOVL C00001 V=800.0 PL=0
MOVL C00002 V=800.0 PL=0
MOVL C00003 V=800.0 PL=0
MOVL C00004 V=800.0 PL=0
MOVL C00005 V=800.0 PL=0
MOVL C00006 V=800.0 PL=0
MOVL C00007 V=800.0 PL=0
MOVL C00008 V=800.0 PL=0
MOVL C00009 V=800.0 PL=0
MOVL C00010 V=800.0 PL=0
MOVL C00011 V=800.0 PL=0
MOVL C00012 V=800.0 PL=0
MOVL C00013 V=800.0 PL=0
MOVL C00014 V=800.0 PL=0
MOVL C00015 V=800.0 PL=0
MOVL C00016 V=800.0 PL=0
MOVL C00017 V=800.0 PL=0
MOVL C00018 V=800.0 PL=0
MOVL C00019 V=800.0 PL=0
MOVL C00020 V=800.0 PL=0
MOVL C00021 V=800.0 PL=0
MOVL C00022 V=800.0 PL=0
MOVL C00023 V=800.0 PL=0
MOVL C00024 V=800.0 PL=0
MOVL C00025 V=800.0 PL=0
MOVL C00026 V=800.0 PL=0
MOVL C00027 V=800.0 PL=0
MOVL C00028 V=800.0 PL=0
MOVL C00029 V=800.0 PL=0
MOVL C00030 V=800.0 PL=0
MOVL C00031 V=800.0 PL=0
MOVL C00032 V=800.0 PL=0
MOVL C00033 V=800.0 PL=0
MOVL C00034 V=800.0 PL=0
MOVL C00035 V=800.0 PL=0
MOVL C00036 V=800.0 PL=0
MOVL C00037 V=800.0 PL=0
MOVL C00038 V=800.0 PL=0
MOVL C00039 V=800.0 PL=0
MOVL C00040 V=800.0 PL=0
MOVL C00041 V=800.0 PL=0
MOVL C00042 V=800.0 PL=0
MOVL C00043 V=800.0 PL=0
MOVL C00044 V=800.0 PL=0
MOVL C00045 V=800.0 PL=0
MOVL C00046 V=800.0 PL=0
MOVL C00047 V=800.0 PL=0
MOVL C00048 V=800.0 PL=0
MOVL C00049 V=800.0 PL=0
MOVL C00050 V=800.0 PL=0
MOVL C00051 V=800.0 PL=0
MOVL C00052 V=800.0 PL=0
MOVL C00053 V=800.0 PL=0
MOVL C00054 V=800.0 PL=0
MOVL C00055 V=800.0 PL=0
MOVL C00056 V=800.0 PL=0
MOVL C00057 V=800.0 PL=0
MOVL C00058 V=800.0 PL=0
MOVL C00059 V=800.0 PL=0
MOVL C00060 V=800.0 PL=0
MOVL C00061 V=800.0 PL=0
MOVL C00062 V=800.0 PL=0
MOVL C00063 V=800.0 PL=0
MOVL C00064 V=800.0 PL=0
MOVL C00065 V=800.0 PL=0
MOVL C00066 V=800.0 PL=0
MOVL C00067 V=800.0 PL=0
MOVL C00068 V=800.0 PL=0
MOVL C00069 V=800.0 PL=0
MOVL C00070 V=800.0 PL=0
MOVL C00071 V=800.0 PL=0
MOVL C00072 V=800.0 PL=0
MOVL C00073 V=800.0 PL=0
MOVL C00074 V=800.0 PL=0
MOVL C00075 V=800.0 PL=0
MOVL C00076 V=800.0 PL=0
MOVL C00077 V=800.0 PL=0
MOVL C00078 V=800.0 PL=0
MOVL C00079 V=800.0 PL=0
MOVL C00080 V=800.0 PL=0
MOVL C00081 V=800.0 PL=0
MOVL C00082 V=800.0 PL=0
MOVL C00083 V=800.0 PL=0
MOVL C00084 V=800.0 PL=0
MOVL C00085 V=800.0 PL=0
MOVL C00086 V=800.0 PL=0
MOVL C00087 V=800.0 PL=0
MOVL C00088 V=800.0 PL=0
MOVL C00089 V=800.0 PL=0
MOVL C00090 V=800.0 PL=0
MOVL C00091 V=800.0 PL=0
MOVL C00092 V=800.0 PL=0
MOVL C00093 V=800.0 PL=0
MOVL C00094 V=800.0 PL=0
MOVL C00095 V=800.0 PL=0
MOVL C00096 V=800.0 PL=0
MOVL C00097 V=800.0 PL=0
MOVL C00098 V=800.0 PL=0
MOVL C00099 V=800.0 PL=0
MOVL C00100 V=800.0 PL=0
MOVL C00101 V=800.0 PL=0
MOVL C00102 V=800.0 PL=0
MOVL C00103 V=800.0 PL=0
MOVL C00104 V=800.0 PL=0
MOVL C00105 V=800.0 PL=0
MOVL C00106 V=800.0 PL=0
MOVL C00107 V=800.0 PL=0
MOVL C00108 V=800.0 PL=0
MOVL C00109 V=800.0 PL=0
MOVL C00110 V=800.0 PL=0
MOVL C00111 V=800.0 PL=0
MOVL C00112 V=800.0 PL=0
MOVL C00113 V=800.0 PL=0
MOVL C00114 V=800.0 PL=0
MOVL C00115 V=800.0 PL=0
MOVL C00116 V=800.0 PL=0
MOVL C00117 V=800.0 PL=0
MOVL C00118 V=800.0 PL=0
MOVL C00119 V=800.0 PL=0
MOVL C00120 V=800.0 PL=0
MOVL C00121 V=800.0 PL=0
MOVL C00122 V=800.0 PL=0
MOVL C00123 V=800.0 PL=0
MOVL C00124 V=800.0 PL=0
MOVL C00125 V=800.0 PL=0
MOVL C00126 V=800.0 PL=0
MOVL C00127 V=800.0 PL=0
MOVL C00128 V=800.0 PL=0
MOVL C00129 V=800.0 PL=0
MOVL C00130 V=800.0 PL=0
MOVL C00131 V=800.0 PL=0
MOVL C00132 V=800.0 PL=0
MOVL C00133 V=800.0 PL=0
MOVL C00134 V=800.0 PL=0
MOVL C00135 V=800.0 PL=0
MOVL C00136 V=800.0 PL=0
MOVL C00137 V=800.0 PL=0
MOVL C00138 V=800.0 PL=0
MOVL C00139 V=800.0 PL=0
MOVL C00140 V=800.0 PL=0
MOVL C00141 V=800.0 PL=0
MOVL C00142 V=800.0 PL=0
MOVL C00143 V=800.0 PL=0
MOVL C00144 V=800.0 PL=0
MOVL C00145 V=800.0 PL=0
MOVL C00146 V=800.0 PL=0
MOVL C00147 V=800.0 PL=0
MOVL C00148 V=800.0 PL=0
MOVL C00149 V=800.0 PL=0
MOVL C00150 V=800.0 PL=0
MOVL C00151 V=800.0 PL=0
MOVL C00152 V=800.0 PL=0
MOVL C00153 V=800.0 PL=0
MOVL C00154 V=800.0 PL=0
MOVL C00155 V=800.0 PL=0
MOVL C00156 V=800.0 PL=0
MOVL C00157 V=800.0 PL=0
MOVL C00158 V=800.0 PL=0
MOVL C00159 V=800.0 PL=0
MOVL C00160 V=800.0 PL=0
MOVL C00161 V=800.0 PL=0
MOVL C00162 V=800.0 PL=0
MOVL C00163 V=800.0 PL=0
MOVL C00164 V=800.0 PL=0
MOVL C00165 V=800.0 PL=0
MOVL C00166 V=800.0 PL=0
MOVL C00167 V=800.0 PL=0
MOVL C00168 V=800.0 PL=0
MOVL C00169 V=800.0 PL=0
MOVL C00170 V=800.0 PL=0
MOVL C00171 V=800.0 PL=0
MOVL C00172 V=800.0 PL=0
MOVL C00173 V=800.0 PL=0
MOVL C00174 V=800.0 PL=0
MOVL C00175 V=800.0 PL=0
MOVL C00176 V=800.0 PL=0
MOVL C00177 V=800.0 PL=0
MOVL C00178 V=800.0 PL=0
MOVL C00179 V=800.0 PL=0
MOVL C00180 V=800.0 PL=0
MOVL C00181 V=800.0 PL=0
MOVL C00182 V=800.0 PL=0
MOVL C00183 V=800.0 PL=0
MOVL C00184 V=800.0 PL=0
MOVL C00185 V=800.0 PL=0
MOVL C00186 V=800.0 PL=0
MOVL C00187 V=800.0 PL=0
MOVL C00188 V=800.0 PL=0
MOVL C00189 V=800.0 PL=0
MOVL C00190 V=800.0 PL=0
MOVL C00191 V=800.0 PL=0
MOVL C00192 V=800.0 PL=0
MOVL C00193 V=800.0 PL=0
MOVL C00194 V=800.0 PL=0
MOVL C00195 V=800.0 PL=0
MOVL C00196 V=800.0 PL=0
MOVL C00197 V=800.0 PL=0
MOVL C00198 V=800.0 PL=0
MOVL C00199 V=800.0 PL=0
MOVL C00200 V=800.0 PL=0
MOVL C00201 V=800.0 PL=0
MOVL C00202 V=800.0 PL=0
MOVL C00203 V=800.0 PL=0
MOVL C00204 V=800.0 PL=0
MOVL C00205 V=800.0 PL=0
MOVL C00206 V=800.0 PL=0
MOVL C00207 V=800.0 PL=0
MOVL C00208 V=800.0 PL=0
MOVL C00209 V=800.0 PL=0
MOVL C00210 V=800.0 PL=0
MOVL C00211 V=800.0 PL=0
MOVL C00212 V=800.0 PL=0
MOVL C00213 V=800.0 PL=0
MOVL C00214 V=800.0 PL=0
MOVL C00215 V=800.0 PL=0
MOVL C00216 V=800.0 PL=0
MOVL C00217 V=800.0 PL=0
MOVL C00218 V=800.0 PL=0
MOVL C00219 V=800.0 PL=0
MOVL C00220 V=800.0 PL=0
MOVL C00221 V=800.0 PL=0
MOVL C00222 V=800.0 PL=0
MOVL C00223 V=800.0 PL=0
MOVL C00224 V=800.0 PL=0
MOVL C00225 V=800.0 PL=0
MOVL C00226 V=800.0 PL=0
MOVL C00227 V=800.0 PL=0
MOVL C00228 V=800.0 PL=0
MOVL C00229 V=800.0 PL=0
MOVL C00230 V=800.0 PL=0
MOVL C00231 V=800.0 PL=0
MOVL C00232 V=800.0 PL=0
MOVL C00233 V=800.0 PL=0
MOVL C00234 V=800.0 PL=0
MOVL C00235 V=800.0 PL=0
MOVL C00236 V=800.0 PL=0
MOVL C00237 V=800.0 PL=0
MOVL C00238 V=800.0 PL=0
MOVL C00239 V=800.0 PL=0
MOVL C00240 V=800.0 PL=0
MOVL C00241 V=800.0 PL=0
MOVL C00242 V=800.0 PL=0
MOVL C00243 V=800.0 PL=0
MOVL C00244 V=800.0 PL=0
MOVL C00245 V=800.0 PL=0
MOVL C00246 V=800.0 PL=0
MOVL C00247 V=800.0 PL=0
MOVL C00248 V=800.0 PL=0
MOVL C00249 V=800.0 PL=0
MOVL C00250 V=800.0 PL=0
MOVL C00251 V=800.0 PL=0
MOVL C00252 V=800.0 PL=0
MOVL C00253 V=800.0 PL=0
MOVL C00254 V=800.0 PL=0
MOVL C00255 V=800.0 PL=0
MOVL C00256 V=800.0 PL=0
MOVL C00257 V=800.0 PL=0
MOVL C00258 V=800.0 PL=0
MOVL C00259 V=800.0 PL=0
MOVL C00260 V=800.0 PL=0
MOVL C00261 V=800.0 PL=0
MOVL C00262 V=800.0 PL=0
MOVL C00263 V=800.0 PL=0
MOVL C00264 V=800.0 PL=0
MOVL C00265 V=800.0 PL=0
MOVL C00266 V=800.0 PL=0
MOVL C00267 V=800.0 PL=0
MOVL C00268 V=800.0 PL=0
MOVL C00269 V=800.0 PL=0
MOVL C00270 V=800.0 PL=0
MOVL C00271 V=800.0 PL=0
MOVL C00272 V=800.0 PL=0
MOVL C00273 V=800.0 PL=0
MOVL C00274 V=800.0 PL=0
MOVL C00275 V=800.0 PL=0
MOVL C00276 V=800.0 PL=0
MOVL C00277 V=800.0 PL=0
MOVL C00278 V=800.0 PL=0
MOVL C00279 V=800.0 PL=0
MOVL C00280 V=800.0 PL=0
MOVL C00281 V=800.0 PL=0
MOVL C00282 V=800.0 PL=0
MOVL C00283 V=800.0 PL=0
MOVL C00284 V=800.0 PL=0
MOVL C00285 V=800.0 PL=0
MOVL C00286 V=800.0 PL=0
MOVL C00287 V=800.0 PL=0
MOVL C00288 V=800.0 PL=0
MOVL C00289 V=800.0 PL=0
MOVL C00290 V=800.0 PL=0
MOVL C00291 V=800.0 PL=0
MOVL C00292 V=800.0 PL=0
MOVL C00293 V=800.0 PL=0
MOVL C00294 V=800.0 PL=0
MOVL C00295 V=800.0 PL=0
MOVL C00296 V=800.0 PL=0
MOVL C00297 V=800.0 PL=0
MOVL C00298 V=800.0 PL=0
MOVL C00299 V=800.0 PL=0
MOVL C00300 V=800.0 PL=0
MOVL C00301 V=800.0 PL=0
MOVL C00302 V=800.0 PL=0
MOVL C00303 V=800.0 PL=0
MOVL C00304 V=800.0 PL=0
MOVL C00305 V=800.0 PL=0
MOVL C00306 V=800.0 PL=0
MOVL C00307 V=800.0 PL=0
MOVL C00308 V=800.0 PL=0
MOVL C00309 V=800.0 PL=0
MOVL C00310 V=800.0 PL=0
MOVL C00311 V=800.0 PL=0
MOVL C00312 V=800.0 PL=0
MOVL C00313 V=800.0 PL=0
MOVL C00314 V=800.0 PL=0
MOVL C00315 V=800.0 PL=0
MOVL C00316 V=800.0 PL=0
MOVL C00317 V=800.0 PL=0
MOVL C00318 V=800.0 PL=0
MOVL C00319 V=800.0 PL=0
MOVL C00320 V=800.0 PL=0
MOVL C00321 V=800.0 PL=0
MOVL C00322 V=800.0 PL=0
MOVL C00323 V=800.0 PL=0
MOVL C00324 V=800.0 PL=0
MOVL C00325 V=800.0 PL=0
MOVL C00326 V=800.0 PL=0
MOVL C00327 V=800.0 PL=0
MOVL C00328 V=800.0 PL=0
MOVL C00329 V=800.0 PL=0
MOVL C00330 V=800.0 PL=0
MOVL C00331 V=800.0 PL=0
MOVL C00332 V=800.0 PL=0
MOVL C00333 V=800.0 PL=0
MOVL C00334 V=800.0 PL=0
MOVL C00335 V=800.0 PL=0
MOVL C00336 V=800.0 PL=0
MOVL C00337 V=800.0 PL=0
MOVL C00338 V=800.0 PL=0
MOVL C00339 V=800.0 PL=0
MOVL C00340 V=800.0 PL=0
MOVL C00341 V=800.0 PL=0
MOVL C00342 V=800.0 PL=0
MOVL C00343 V=800.0 PL=0
MOVL C00344 V=800.0 PL=0
MOVL C00345 V=800.0 PL=0
MOVL C00346 V=800.0 PL=0
MOVL C00347 V=800.0 PL=0
MOVL C00348 V=800.0 PL=0
MOVL C00349 V=800.0 PL=0
MOVL C00350 V=800.0 PL=0
MOVL C00351 V=800.0 PL=0
MOVL C00352 V=800.0 PL=0
MOVL C00353 V=800.0 PL=0
MOVL C00354 V=800.0 PL=0
MOVL C00355 V=800.0 PL=0
MOVL C00356 V=800.0 PL=0
MOVL C00357 V=800.0 PL=0
MOVL C00358 V=800.0 PL=0
MOVL C00359 V=800.0 PL=0
MOVL C00360 V=800.0 PL=0
MOVL C00361 V=800.0 PL=0
MOVL C00362 V=800.0 PL=0
MOVL C00363 V=800.0 PL=0
MOVL C00364 V=800.0 PL=0
MOVL C00365 V=800.0 PL=0
MOVL C00366 V=800.0 PL=0
MOVL C00367 V=800.0 PL=0
MOVL C00368 V=800.0 PL=0
MOVL C00369 V=800.0 PL=0
MOVL C00370 V=800.0 PL=0
MOVL C00371 V=800.0 PL=0
MOVL C00372 V=800.0 PL=0
MOVL C00373 V=800.0 PL=0
MOVL C00374 V=800.0 PL=0
MOVL C00375 V=800.0 PL=0
MOVL C00376 V=800.0 PL=0
MOVL C00377 V=800.0 PL=0
MOVL C00378 V=800.0 PL=0
MOVL C00379 V=800.0 PL=0
MOVL C00380 V=800.0 PL=0
MOVL C00381 V=800.0 PL=0
MOVL C00382 V=800.0 PL=0
MOVL C00383 V=800.0 PL=0
MOVL C00384 V=800.0 PL=0
MOVL C00385 V=800.0 PL=0
MOVL C00386 V=800.0 PL=0
MOVL C00387 V=800.0 PL=0
MOVL C00388 V=800.0 PL=0
MOVL C00389 V=800.0 PL=0
MOVL C00390 V=800.0 PL=0
MOVL C00391 V=800.0 PL=0
MOVL C00392 V=800.0 PL=0
MOVL C00393 V=800.0 PL=0
MOVL C00394 V=800.0 PL=0
MOVL C00395 V=800.0 PL=0
MOVL C00396 V=800.0 PL=0
MOVL C00397 V=800.0 PL=0
MOVL C00398 V=800.0 PL=0
MOVL C00399 V=800.0 PL=0
MOVL C00400 V=800.0 PL=0
MOVL C00401 V=800.0 PL=0
MOVL C00402 V=800.0 PL=0
MOVL C00403 V=800.0 PL=0
MOVL C00404 V=800.0 PL=0
MOVL C00405 V=800.0 PL=0
MOVL C00406 V=800.0 PL=0
MOVL C00407 V=800.0 PL=0
MOVL C00408 V=800.0 PL=0
MOVL C00409 V=800.0 PL=0
MOVL C00410 V=800.0 PL=0
MOVL C00411 V=800.0 PL=0
MOVL C00412 V=800.0 PL=0
MOVL C00413 V=800.0 PL=0
MOVL C00414 V=800.0 PL=0
MOVL C00415 V=800.0 PL=0
MOVL C00416 V=800.0 PL=0
MOVL C00417 V=800.0 PL=0
MOVL C00418 V=800.0 PL=0
MOVL C00419 V=800.0 PL=0
MOVL C00420 V=800.0 PL=0
MOVL C00421 V=800.0 PL=0
MOVL C00422 V=800.0 PL=0
MOVL C00423 V=800.0 PL=0
MOVL C00424 V=800.0 PL=0
MOVL C00425 V=800.0 PL=0
MOVL C00426 V=800.0 PL=0
MOVL C00427 V=800.0 PL=0
MOVL C00428 V=800.0 PL=0
MOVL C00429 V=800.0 PL=0
MOVL C00430 V=800.0 PL=0
MOVL C00431 V=800.0 PL=0
MOVL C00432 V=800.0 PL=0
MOVL C00433 V=800.0 PL=0
MOVL C00434 V=800.0 PL=0
MOVL C00435 V=800.0 PL=0
MOVL C00436 V=800.0 PL=0
MOVL C00437 V=800.0 PL=0
MOVL C00438 V=800.0 PL=0
MOVL C00439 V=800.0 PL=0
MOVL C00440 V=800.0 PL=0
MOVL C00441 V=800.0 PL=0
MOVL C00442 V=800.0 PL=0
MOVL C00443 V=800.0 PL=0
MOVL C00444 V=800.0 PL=0
MOVL C00445 V=800.0 PL=0
MOVL C00446 V=800.0 PL=0
MOVL C00447 V=800.0 PL=0
MOVL C00448 V=800.0 PL=0
MOVL C00449 V=800.0 PL=0
MOVL C00450 V=800.0 PL=0
MOVL C00451 V=800.0 PL=0
MOVL C00452 V=800.0 PL=0
MOVL C00453 V=800.0 PL=0
MOVL C00454 V=800.0 PL=0
MOVL C00455 V=800.0 PL=0
MOVL C00456 V=800.0 PL=0
MOVL C00457 V=800.0 PL=0
MOVL C00458 V=800.0 PL=0
MOVL C00459 V=800.0 PL=0
MOVL C00460 V=800.0 PL=0
MOVL C00461 V=800.0 PL=0
MOVL C00462 V=800.0 PL=0
MOVL C00463 V=800.0 PL=0
MOVL C00464 V=800.0 PL=0
MOVL C00465 V=800.0 PL=0
MOVL C00466 V=800.0 PL=0
MOVL C00467 V=800.0 PL=0
MOVL C00468 V=800.0 PL=0
MOVL C00469 V=800.0 PL=0
MOVL C00470 V=800.0 PL=0
MOVL C00471 V=800.0 PL=0
MOVL C00472 V=800.0 PL=0
MOVL C00473 V=800.0 PL=0
MOVL C00474 V=800.0 PL=0
MOVL C00475 V=800.0 PL=0
MOVL C00476 V=800.0 PL=0
MOVL C00477 V=800.0 PL=0
MOVL C00478 V=800.0 PL=0
MOVL C00479 V=800.0 PL=0
MOVL C00480 V=800.0 PL=0
MOVL C00481 V=800.0 PL=0
MOVL C00482 V=800.0 PL=0
MOVL C00483 V=800.0 PL=0
MOVL C00484 V=800.0 PL=0
MOVL C00485 V=800.0 PL=0
MOVL C00486 V=800.0 PL=0
MOVL C00487 V=800.0 PL=0
MOVL C00488 V=800.0 PL=0
MOVL C00489 V=800.0 PL=0
MOVL C00490 V=800.0 PL=0
MOVL C00491 V=800.0 PL=0
MOVL C00492 V=800.0 PL=0
MOVL C00493 V=800.0 PL=0
MOVL C00494 V=800.0 PL=0
MOVL C00495 V=800.0 PL=0
MOVL C00496 V=800.0 PL=0
MOVL C00497 V=800.0 PL=0
MOVL C00498 V=800.0 PL=0
MOVL C00499 V=800.0 PL=0
MOVL C00500 V=800.0 PL=0
MOVL C00501 V=800.0 PL=0
MOVL C00502 V=800.0 PL=0
MOVL C00503 V=800.0 PL=0
MOVL C00504 V=800.0 PL=0
MOVL C00505 V=800.0 PL=0
MOVL C00506 V=800.0 PL=0
MOVL C00507 V=800.0 PL=0
MOVL C00508 V=800.0 PL=0
MOVL C00509 V=800.0 PL=0
MOVL C00510 V=800.0 PL=0
MOVL C00511 V=800.0 PL=0
MOVL C00512 V=800.0 PL=0
MOVL C00513 V=800.0 PL=0
MOVL C00514 V=800.0 PL=0
MOVL C00515 V=800.0 PL=0
MOVL C00516 V=800.0 PL=0
MOVL C00517 V=800.0 PL=0
MOVL C00518 V=800.0 PL=0
MOVL C00519 V=800.0 PL=0
MOVL C00520 V=800.0 PL=0
MOVL C00521 V=800.0 PL=0
MOVL C00522 V=800.0 PL=0
MOVL C00523 V=800.0 PL=0
MOVL C00524 V=800.0 PL=0
MOVL C00525 V=800.0 PL=0
MOVL C00526 V=800.0 PL=0
MOVL C00527 V=800.0 PL=0
MOVL C00528 V=800.0 PL=0
MOVL C00529 V=800.0 PL=0
MOVL C00530 V=800.0 PL=0
MOVL C00531 V=800.0 PL=0
MOVL C00532 V=800.0 PL=0
MOVL C00533 V=800.0 PL=0
MOVL C00534 V=800.0 PL=0
MOVL C00535 V=800.0 PL=0
MOVL C00536 V=800.0 PL=0
MOVL C00537 V=800.0 PL=0
MOVL C00538 V=800.0 PL=0
MOVL C00539 V=800.0 PL=0
MOVL C00540 V=800.0 PL=0
MOVL C00541 V=800.0 PL=0
MOVL C00542 V=800.0 PL=0
MOVL C00543 V=800.0 PL=0
MOVL C00544 V=800.0 PL=0
MOVL C00545 V=800.0 PL=0
MOVL C00546 V=800.0 PL=0
MOVL C00547 V=800.0 PL=0
MOVL C00548 V=800.0 PL=0
MOVL C00549 V=800.0 PL=0
MOVL C00550 V=800.0 PL=0
MOVL C00551 V=800.0 PL=0
MOVL C00552 V=800.0 PL=0
MOVL C00553 V=800.0 PL=0
MOVL C00554 V=800.0 PL=0
MOVL C00555 V=800.0 PL=0
MOVL C00556 V=800.0 PL=0
MOVL C00557 V=800.0 PL=0
MOVL C00558 V=800.0 PL=0
MOVL C00559 V=800.0 PL=0
MOVL C00560 V=800.0 PL=0
MOVL C00561 V=800.0 PL=0
MOVL C00562 V=800.0 PL=0
MOVL C00563 V=800.0 PL=0
MOVL C00564 V=800.0 PL=0
MOVL C00565 V=800.0 PL=0
MOVL C00566 V=800.0 PL=0
MOVL C00567 V=800.0 PL=0
MOVL C00568 V=800.0 PL=0
MOVL C00569 V=800.0 PL=0
MOVL C00570 V=800.0 PL=0
MOVL C00571 V=800.0 PL=0
MOVL C00572 V=800.0 PL=0
MOVL C00573 V=800.0 PL=0
MOVL C00574 V=800.0 PL=0
MOVL C00575 V=800.0 PL=0
MOVL C00576 V=800.0 PL=0
MOVL C00577 V=800.0 PL=0
MOVL C00578 V=800.0 PL=0
MOVL C00579 V=800.0 PL=0
MOVL C00580 V=800.0 PL=0
MOVL C00581 V=800.0 PL=0
MOVL C00582 V=800.0 PL=0
MOVL C00583 V=800.0 PL=0
MOVL C00584 V=800.0 PL=0
MOVL C00585 V=800.0 PL=0
MOVL C00586 V=800.0 PL=0
MOVL C00587 V=800.0 PL=0
MOVL C00588 V=800.0 PL=0
MOVL C00589 V=800.0 PL=0
MOVL C00590 V=800.0 PL=0
MOVL C00591 V=800.0 PL=0
MOVL C00592 V=800.0 PL=0
MOVL C00593 V=800.0 PL=0
MOVL C00594 V=800.0 PL=0
MOVL C00595 V=800.0 PL=0
MOVL C00596 V=800.0 PL=0
MOVL C00597 V=800.0 PL=0
MOVL C00598 V=800.0 PL=0
MOVL C00599 V=800.0 PL=0
MOVL C00600 V=800.0 PL=0
MOVL C00601 V=800.0 PL=0
MOVL C00602 V=800.0 PL=0
MOVL C00603 V=800.0 PL=0
MOVL C00604 V=800.0 PL=0
MOVL C00605 V=800.0 PL=0
MOVL C00606 V=800.0 PL=0
MOVL C00607 V=800.0 PL=0
MOVL C00608 V=800.0 PL=0
MOVL C00609 V=800.0 PL=0
MOVL C00610 V=800.0 PL=0
MOVL C00611 V=800.0 PL=0
MOVL C00612 V=800.0 PL=0
MOVL C00613 V=800.0 PL=0
MOVL C00614 V=800.0 PL=0
MOVL C00615 V=800.0 PL=0
MOVL C00616 V=800.0 PL=0
MOVL C00617 V=800.0 PL=0
MOVL C00618 V=800.0 PL=0
MOVL C00619 V=800.0 PL=0
MOVL C00620 V=800.0 PL=0
MOVL C00621 V=800.0 PL=0
MOVL C00622 V=800.0 PL=0
MOVL C00623 V=800.0 PL=0
MOVL C00624 V=800.0 PL=0
MOVL C00625 V=800.0 PL=0
MOVL C00626 V=800.0 PL=0
MOVL C00627 V=800.0 PL=0
MOVL C00628 V=800.0 PL=0
MOVL C00629 V=800.0 PL=0
MOVL C00630 V=800.0 PL=0
MOVL C00631 V=800.0 PL=0
MOVL C00632 V=800.0 PL=0
MOVL C00633 V=800.0 PL=0
MOVL C00634 V=800.0 PL=0
MOVL C00635 V=800.0 PL=0
MOVL C00636 V=800.0 PL=0
MOVL C00637 V=800.0 PL=0
MOVL C00638 V=800.0 PL=0
MOVL C00639 V=800.0 PL=0
MOVL C00640 V=800.0 PL=0
MOVL C00641 V=800.0 PL=0
MOVL C00642 V=800.0 PL=0
MOVL C00643 V=800.0 PL=0
MOVL C00644 V=800.0 PL=0
MOVL C00645 V=800.0 PL=0
MOVL C00646 V=800.0 PL=0
MOVL C00647 V=800.0 PL=0
MOVL C00648 V=800.0 PL=0
MOVL C00649 V=800.0 PL=0
MOVL C00650 V=800.0 PL=0
MOVL C00651 V=800.0 PL=0
MOVL C00652 V=800.0 PL=0
MOVL C00653 V=800.0 PL=0
MOVL C00654 V=800.0 PL=0
MOVL C00655 V=800.0 PL=0
MOVL C00656 V=800.0 PL=0
MOVL C00657 V=800.0 PL=0
MOVL C00658 V=800.0 PL=0
MOVL C00659 V=800.0 PL=0
MOVL C00660 V=800.0 PL=0
MOVL C00661 V=800.0 PL=0
MOVL C00662 V=800.0 PL=0
MOVL C00663 V=800.0 PL=0
MOVL C00664 V=800.0 PL=0
MOVL C00665 V=800.0 PL=0
MOVL C00666 V=800.0 PL=0
MOVL C00667 V=800.0 PL=0
MOVL C00668 V=800.0 PL=0
MOVL C00669 V=800.0 PL=0
MOVL C00670 V=800.0 PL=0
MOVL C00671 V=800.0 PL=0
MOVL C00672 V=800.0 PL=0
MOVL C00673 V=800.0 PL=0
MOVL C00674 V=800.0 PL=0
MOVL C00675 V=800.0 PL=0
MOVL C00676 V=800.0 PL=0
MOVL C00677 V=800.0 PL=0
MOVL C00678 V=800.0 PL=0
MOVL C00679 V=800.0 PL=0
MOVL C00680 V=800.0 PL=0
MOVL C00681 V=800.0 PL=0
MOVL C00682 V=800.0 PL=0
MOVL C00683 V=800.0 PL=0
MOVL C00684 V=800.0 PL=0
MOVL C00685 V=800.0 PL=0
MOVL C00686 V=800.0 PL=0
MOVL C00687 V=800.0 PL=0
MOVL C00688 V=800.0 PL=0
MOVL C00689 V=800.0 PL=0
MOVL C00690 V=800.0 PL=0
MOVL C00691 V=800.0 PL=0
MOVL C00692 V=800.0 PL=0
MOVL C00693 V=800.0 PL=0
MOVL C00694 V=800.0 PL=0
MOVL C00695 V=800.0 PL=0
MOVL C00696 V=800.0 PL=0
MOVL C00697 V=800.0 PL=0
MOVL C00698 V=800.0 PL=0
MOVL C00699 V=800.0 PL=0
MOVL C00700 V=800.0 PL=0
MOVL C00701 V=800.0 PL=0
MOVL C00702 V=800.0 PL=0
MOVL C00703 V=800.0 PL=0
MOVL C00704 V=800.0 PL=0
MOVL C00705 V=800.0 PL=0
MOVL C00706 V=800.0 PL=0
MOVL C00707 V=800.0 PL=0
MOVL C00708 V=800.0 PL=0
MOVL C00709 V=800.0 PL=0
MOVL C00710 V=800.0 PL=0
MOVL C00711 V=800.0 PL=0
MOVL C00712 V=800.0 PL=0
MOVL C00713 V=800.0 PL=0
MOVL C00714 V=800.0 PL=0
MOVL C00715 V=800.0 PL=0
MOVL C00716 V=800.0 PL=0
MOVL C00717 V=800.0 PL=0
MOVL C00718 V=800.0 PL=0
MOVL C00719 V=800.0 PL=0
MOVL C00720 V=800.0 PL=0
MOVL C00721 V=800.0 PL=0
MOVL C00722 V=800.0 PL=0
MOVL C00723 V=800.0 PL=0
MOVL C00724 V=800.0 PL=0
MOVL C00725 V=800.0 PL=0
MOVL C00726 V=800.0 PL=0
MOVL C00727 V=800.0 PL=0
MOVL C00728 V=800.0 PL=0
MOVL C00729 V=800.0 PL=0
MOVL C00730 V=800.0 PL=0
MOVL C00731 V=800.0 PL=0
MOVL C00732 V=800.0 PL=0
MOVL C00733 V=800.0 PL=0
MOVL C00734 V=800.0 PL=0
MOVL C00735 V=800.0 PL=0
MOVL C00736 V=800.0 PL=0
MOVL C00737 V=800.0 PL=0
MOVL C00738 V=800.0 PL=0
MOVL C00739 V=800.0 PL=0
MOVL C00740 V=800.0 PL=0
MOVL C00741 V=800.0 PL=0
MOVL C00742 V=800.0 PL=0
MOVL C00743 V=800.0 PL=0
MOVL C00744 V=800.0 PL=0
MOVL C00745 V=800.0 PL=0
MOVL C00746 V=800.0 PL=0
MOVL C00747 V=800.0 PL=0
MOVL C00748 V=800.0 PL=0
MOVL C00749 V=800.0 PL=0
MOVL C00750 V=800.0 PL=0
MOVL C00751 V=800.0 PL=0
MOVL C00752 V=800.0 PL=0
MOVL C00753 V=800.0 PL=0
MOVL C00754 V=800.0 PL=0
MOVL C00755 V=800.0 PL=0
MOVL C00756 V=800.0 PL=0
MOVL C00757 V=800.0 PL=0
MOVL C00758 V=800.0 PL=0
MOVL C00759 V=800.0 PL=0
MOVL C00760 V=800.0 PL=0
MOVL C00761 V=800.0 PL=0
MOVL C00762 V=800.0 PL=0
MOVL C00763 V=800.0 PL=0
MOVL C00764 V=800.0 PL=0
MOVL C00765 V=800.0 PL=0
MOVL C00766 V=800.0 PL=0
MOVL C00767 V=800.0 PL=0
MOVL C00768 V=800.0 PL=0
MOVL C00769 V=800.0 PL=0
MOVL C00770 V=800.0 PL=0
MOVL C00771 V=800.0 PL=0
MOVL C00772 V=800.0 PL=0
MOVL C00773 V=800.0 PL=0
MOVL C00774 V=800.0 PL=0
MOVL C00775 V=800.0 PL=0
MOVL C00776 V=800.0 PL=0
MOVL C00777 V=800.0 PL=0
MOVL C00778 V=800.0 PL=0
MOVL C00779 V=800.0 PL=0
MOVL C00780 V=800.0 PL=0
MOVL C00781 V=800.0 PL=0
MOVL C00782 V=800.0 PL=0
MOVL C00783 V=800.0 PL=0
MOVL C00784 V=800.0 PL=0
MOVL C00785 V=800.0 PL=0
MOVL C00786 V=800.0 PL=0
MOVL C00787 V=800.0 PL=0
MOVL C00788 V=800.0 PL=0
MOVL C00789 V=800.0 PL=0
MOVL C00790 V=800.0 PL=0
MOVL C00791 V=800.0 PL=0
MOVL C00792 V=800.0 PL=0
MOVL C00793 V=800.0 PL=0
MOVL C00794 V=800.0 PL=0
MOVL C00795 V=800.0 PL=0
MOVL C00796 V=800.0 PL=0
MOVL C00797 V=800.0 PL=0
MOVL C00798 V=800.0 PL=0
MOVL C00799 V=800.0 PL=0
MOVL C00800 V=800.0 PL=0
MOVL C00801 V=800.0 PL=0
MOVL C00802 V=800.0 PL=0
MOVL C00803 V=800.0 PL=0
MOVL C00804 V=800.0 PL=0
MOVL C00805 V=800.0 PL=0
MOVL C00806 V=800.0 PL=0
MOVL C00807 V=800.0 PL=0
MOVL C00808 V=800.0 PL=0
MOVL C00809 V=800.0 PL=0
MOVL C00810 V=800.0 PL=0
MOVL C00811 V=800.0 PL=0
MOVL C00812 V=800.0 PL=0
MOVL C00813 V=800.0 PL=0
MOVL C00814 V=800.0 PL=0
MOVL C00815 V=800.0 PL=0
MOVL C00816 V=800.0 PL=0
MOVL C00817 V=800.0 PL=0
MOVL C00818 V=800.0 PL=0
MOVL C00819 V=800.0 PL=0
MOVL C00820 V=800.0 PL=0
MOVL C00821 V=800.0 PL=0
MOVL C00822 V=800.0 PL=0
MOVL C00823 V=800.0 PL=0
MOVL C00824 V=800.0 PL=0
MOVL C00825 V=800.0 PL=0
MOVL C00826 V=800.0 PL=0
MOVL C00827 V=800.0 PL=0
MOVL C00828 V=800.0 PL=0
MOVL C00829 V=800.0 PL=0
MOVL C00830 V=800.0 PL=0
MOVL C00831 V=800.0 PL=0
MOVL C00832 V=800.0 PL=0
MOVL C00833 V=800.0 PL=0
MOVL C00834 V=800.0 PL=0
MOVL C00835 V=800.0 PL=0
MOVL C00836 V=800.0 PL=0
MOVL C00837 V=800.0 PL=0
MOVL C00838 V=800.0 PL=0
MOVL C00839 V=800.0 PL=0
MOVL C00840 V=800.0 PL=0
MOVL C00841 V=800.0 PL=0
MOVL C00842 V=800.0 PL=0
MOVL C00843 V=800.0 PL=0
MOVL C00844 V=800.0 PL=0
MOVL C00845 V=800.0 PL=0
MOVL C00846 V=800.0 PL=0
MOVL C00847 V=800.0 PL=0
MOVL C00848 V=800.0 PL=0
MOVL C00849 V=800.0 PL=0
MOVL C00850 V=800.0 PL=0
MOVL C00851 V=800.0 PL=0
MOVL C00852 V=800.0 PL=0
MOVL C00853 V=800.0 PL=0
MOVL C00854 V=800.0 PL=0
MOVL C00855 V=800.0 PL=0
MOVL C00856 V=800.0 PL=0
MOVL C00857 V=800.0 PL=0
MOVL C00858 V=800.0 PL=0
MOVL C00859 V=800.0 PL=0
MOVL C00860 V=800.0 PL=0
MOVL C00861 V=800.0 PL=0
MOVL C00862 V=800.0 PL=0
MOVL C00863 V=800.0 PL=0
MOVL C00864 V=800.0 PL=0
MOVL C00865 V=800.0 PL=0
MOVL C00866 V=800.0 PL=0
MOVL C00867 V=800.0 PL=0
MOVL C00868 V=800.0 PL=0
MOVL C00869 V=800.0 PL=0
MOVL C00870 V=800.0 PL=0
MOVL C00871 V=800.0 PL=0
MOVL C00872 V=800.0 PL=0
MOVL C00873 V=800.0 PL=0
MOVL C00874 V=800.0 PL=0
MOVL C00875 V=800.0 PL=0
MOVL C00876 V=800.0 PL=0
MOVL C00877 V=800.0 PL=0
MOVL C00878 V=800.0 PL=0
MOVL C00879 V=800.0 PL=0
MOVL C00880 V=800.0 PL=0
MOVL C00881 V=800.0 PL=0
MOVL C00882 V=800.0 PL=0
MOVL C00883 V=800.0 PL=0
MOVL C00884 V=800.0 PL=0
MOVL C00885 V=800.0 PL=0
MOVL C00886 V=800.0 PL=0
MOVL C00887 V=800.0 PL=0
MOVL C00888 V=800.0 PL=0
MOVL C00889 V=800.0 PL=0
MOVL C00890 V=800.0 PL=0
MOVL C00891 V=800.0 PL=0
MOVL C00892 V=800.0 PL=0
MOVL C00893 V=800.0 PL=0
MOVL C00894 V=800.0 PL=0
MOVL C00895 V=800.0 PL=0
MOVL C00896 V=800.0 PL=0
MOVL C00897 V=800.0 PL=0
MOVL C00898 V=800.0 PL=0
MOVL C00899 V=800.0 PL=0
MOVL C00900 V=800.0 PL=0
MOVL C00901 V=800.0 PL=0
MOVL C00902 V=800.0 PL=0
MOVL C00903 V=800.0 PL=0
MOVL C00904 V=800.0 PL=0
MOVL C00905 V=800.0 PL=0
MOVL C00906 V=800.0 PL=0
MOVL C00907 V=800.0 PL=0
MOVL C00908 V=800.0 PL=0
MOVL C00909 V=800.0 PL=0
MOVL C00910 V=800.0 PL=0
MOVL C00911 V=800.0 PL=0
MOVL C00912 V=800.0 PL=0
MOVL C00913 V=800.0 PL=0
MOVL C00914 V=800.0 PL=0
MOVL C00915 V=800.0 PL=0
MOVL C00916 V=800.0 PL=0
MOVL C00917 V=800.0 PL=0
MOVL C00918 V=800.0 PL=0
MOVL C00919 V=800.0 PL=0
MOVL C00920 V=800.0 PL=0
MOVL C00921 V=800.0 PL=0
MOVL C00922 V=800.0 PL=0
MOVL C00923 V=800.0 PL=0
MOVL C00924 V=800.0 PL=0
MOVL C00925 V=800.0 PL=0
MOVL C00926 V=800.0 PL=0
MOVL C00927 V=800.0 PL=0
MOVL C00928 V=800.0 PL=0
MOVL C00929 V=800.0 PL=0
MOVL C00930 V=800.0 PL=0
MOVL C00931 V=800.0 PL=0
MOVL C00932 V=800.0 PL=0
MOVL C00933 V=800.0 PL=0
MOVL C00934 V=800.0 PL=0
MOVL C00935 V=800.0 PL=0
MOVL C00936 V=800.0 PL=0
MOVL C00937 V=800.0 PL=0
MOVL C00938 V=800.0 PL=0
MOVL C00939 V=800.0 PL=0
MOVL C00940 V=800.0 PL=0
MOVL C00941 V=800.0 PL=0
MOVL C00942 V=800.0 PL=0
MOVL C00943 V=800.0 PL=0
MOVL C00944 V=800.0 PL=0
MOVL C00945 V=800.0 PL=0
MOVL C00946 V=800.0 PL=0
MOVL C00947 V=800.0 PL=0
MOVL C00948 V=800.0 PL=0
MOVL C00949 V=800.0 PL=0
MOVL C00950 V=800.0 PL=0
MOVL C00951 V=800.0 PL=0
MOVL C00952 V=800.0 PL=0
MOVL C00953 V=800.0 PL=0
MOVL C00954 V=800.0 PL=0
MOVL C00955 V=800.0 PL=0
MOVL C00956 V=800.0 PL=0
MOVL C00957 V=800.0 PL=0
MOVL C00958 V=800.0 PL=0
MOVL C00959 V=800.0 PL=0
MOVL C00960 V=800.0 PL=0
MOVL C00961 V=800.0 PL=0
MOVL C00962 V=800.0 PL=0
MOVL C00963 V=800.0 PL=0
MOVL C00964 V=800.0 PL=0
MOVL C00965 V=800.0 PL=0
MOVL C00966 V=800.0 PL=0
MOVL C00967 V=800.0 PL=0
MOVL C00968 V=800.0 PL=0
MOVL C00969 V=800.0 PL=0
MOVL C00970 V=800.0 PL=0
MOVL C00971 V=800.0 PL=0
MOVL C00972 V=800.0 PL=0
MOVL C00973 V=800.0 PL=0
MOVL C00974 V=800.0 PL=0
MOVL C00975 V=800.0 PL=0
MOVL C00976 V=800.0 PL=0
MOVL C00977 V=800.0 PL=0
MOVL C00978 V=800.0 PL=0
MOVL C00979 V=800.0 PL=0
MOVL C00980 V=800.0 PL=0
MOVL C00981 V=800.0 PL=0
MOVL C00982 V=800.0 PL=0
MOVL C00983 V=800.0 PL=0
MOVL C00984 V=800.0 PL=0
MOVL C00985 V=800.0 PL=0
MOVL C00986 V=800.0 PL=0
MOVL C00987 V=800.0 PL=0
MOVL C00988 V=800.0 PL=0
MOVL C00989 V=800.0 PL=0
MOVL C00990 V=800.0 PL=0
MOVL C00991 V=800.0 PL=0
MOVL C00992 V=800.0 PL=0
MOVL C00993 V=800.0 PL=0
MOVL C00994 V=800.0 PL=0
MOVL C00995 V=800.0 PL=0
MOVL C00996 V=800.0 PL=0
MOVL C00997 V=800.0 PL=0
MOVL C00998 V=800.0 PL=0
MOVL C00999 V=800.0 PL=0
MOVL C01000 V=800.0 PL=0
MOVL C01001 V=800.0 PL=0
MOVL C01002 V=800.0 PL=0
MOVL C01003 V=800.0 PL=0
MOVL C01004 V=800.0 PL=0
MOVL C01005 V=800.0 PL=0
MOVL C01006 V=800.0 PL=0
MOVL C01007 V=800.0 PL=0
MOVL C01008 V=800.0 PL=0
MOVL C01009 V=800.0 PL=0
MOVL C01010 V=800.0 PL=0
MOVL C01011 V=800.0 PL=0
MOVL C01012 V=800.0 PL=0
MOVL C01013 V=800.0 PL=0
MOVL C01014 V=800.0 PL=0
MOVL C01015 V=800.0 PL=0
MOVL C01016 V=800.0 PL=0
MOVL C01017 V=800.0 PL=0
MOVL C01018 V=800.0 PL=0
MOVL C01019 V=800.0 PL=0
MOVL C01020 V=800.0 PL=0
MOVL C01021 V=800.0 PL=0
MOVL C01022 V=800.0 PL=0
MOVL C01023 V=800.0 PL=0
MOVL C01024 V=800.0 PL=0
MOVL C01025 V=800.0 PL=0
MOVL C01026 V=800.0 PL=0
MOVL C01027 V=800.0 PL=0
MOVL C01028 V=800.0 PL=0
MOVL C01029 V=800.0 PL=0
MOVL C01030 V=800.0 PL=0
MOVL C01031 V=800.0 PL=0
MOVL C01032 V=800.0 PL=0
MOVL C01033 V=800.0 PL=0
MOVL C01034 V=800.0 PL=0
MOVL C01035 V=800.0 PL=0
MOVL C01036 V=800.0 PL=0
MOVL C01037 V=800.0 PL=0
MOVL C01038 V=800.0 PL=0
MOVL C01039 V=800.0 PL=0
MOVL C01040 V=800.0 PL=0
MOVL C01041 V=800.0 PL=0
MOVL C01042 V=800.0 PL=0
MOVL C01043 V=800.0 PL=0
MOVL C01044 V=800.0 PL=0
MOVL C01045 V=800.0 PL=0
MOVL C01046 V=800.0 PL=0
MOVL C01047 V=800.0 PL=0
MOVL C01048 V=800.0 PL=0
MOVL C01049 V=800.0 PL=0
MOVL C01050 V=800.0 PL=0
MOVL C01051 V=800.0 PL=0
MOVL C01052 V=800.0 PL=0
MOVL C01053 V=800.0 PL=0
MOVL C01054 V=800.0 PL=0
MOVL C01055 V=800.0 PL=0
MOVL C01056 V=800.0 PL=0
MOVL C01057 V=800.0 PL=0
MOVL C01058 V=800.0 PL=0
MOVL C01059 V=800.0 PL=0
MOVL C01060 V=800.0 PL=0
MOVL C01061 V=800.0 PL=0
MOVL C01062 V=800.0 PL=0
MOVL C01063 V=800.0 PL=0
MOVL C01064 V=800.0 PL=0
MOVL C01065 V=800.0 PL=0
MOVL C01066 V=800.0 PL=0
MOVL C01067 V=800.0 PL=0
MOVL C01068 V=800.0 PL=0
MOVL C01069 V=800.0 PL=0
MOVL C01070 V=800.0 PL=0
MOVL C01071 V=800.0 PL=0
MOVL C01072 V=800.0 PL=0
MOVL C01073 V=800.0 PL=0
MOVL C01074 V=800.0 PL=0
MOVL C01075 V=800.0 PL=0
MOVL C01076 V=800.0 PL=0
MOVL C01077 V=800.0 PL=0
MOVL C01078 V=800.0 PL=0
MOVL C01079 V=800.0 PL=0
MOVL C01080 V=800.0 PL=0
MOVL C01081 V=800.0 PL=0
MOVL C01082 V=800.0 PL=0
MOVL C01083 V=800.0 PL=0
MOVL C01084 V=800.0 PL=0
MOVL C01085 V=800.0 PL=0
MOVL C01086 V=800.0 PL=0
MOVL C01087 V=800.0 PL=0
MOVL C01088 V=800.0 PL=0
MOVL C01089 V=800.0 PL=0
MOVL C01090 V=800.0 PL=0
MOVL C01091 V=800.0 PL=0
MOVL C01092 V=800.0 PL=0
MOVL C01093 V=800.0 PL=0
MOVL C01094 V=800.0 PL=0
MOVL C01095 V=800.0 PL=0
MOVL C01096 V=800.0 PL=0
MOVL C01097 V=800.0 PL=0
MOVL C01098 V=800.0 PL=0
MOVL C01099 V=800.0 PL=0
MOVL C01100 V=800.0 PL=0
MOVL C01101 V=800.0 PL=0
MOVL C01102 V=800.0 PL=0
MOVL C01103 V=800.0 PL=0
MOVL C01104 V=800.0 PL=0
MOVL C01105 V=800.0 PL=0
MOVL C01106 V=800.0 PL=0
MOVL C01107 V=800.0 PL=0
MOVL C01108 V=800.0 PL=0
MOVL C01109 V=800.0 PL=0
MOVL C01110 V=800.0 PL=0
MOVL C01111 V=800.0 PL=0
MOVL C01112 V=800.0 PL=0
MOVL C01113 V=800.0 PL=0
MOVL C01114 V=800.0 PL=0
MOVL C01115 V=800.0 PL=0
MOVL C01116 V=800.0 PL=0
MOVL C01117 V=800.0 PL=0
MOVL C01118 V=800.0 PL=0
MOVL C01119 V=800.0 PL=0
MOVL C01120 V=800.0 PL=0
MOVL C01121 V=800.0 PL=0
MOVL C01122 V=800.0 PL=0
MOVL C01123 V=800.0 PL=0
MOVL C01124 V=800.0 PL=0
MOVL C01125 V=800.0 PL=0
MOVL C01126 V=800.0 PL=0
MOVL C01127 V=800.0 PL=0
MOVL C01128 V=800.0 PL=0
MOVL C01129 V=800.0 PL=0
MOVL C01130 V=800.0 PL=0
MOVL C01131 V=800.0 PL=0
MOVL C01132 V=800.0 PL=0
MOVL C01133 V=800.0 PL=0
MOVL C01134 V=800.0 PL=0
MOVL C01135 V=800.0 PL=0
MOVL C01136 V=800.0 PL=0
MOVL C01137 V=800.0 PL=0
MOVL C01138 V=800.0 PL=0
MOVL C01139 V=800.0 PL=0
MOVL C01140 V=800.0 PL=0
MOVL C01141 V=800.0 PL=0
MOVL C01142 V=800.0 PL=0
MOVL C01143 V=800.0 PL=0
MOVL C01144 V=800.0 PL=0
MOVL C01145 V=800.0 PL=0
MOVL C01146 V=800.0 PL=0
MOVL C01147 V=800.0 PL=0
MOVL C01148 V=800.0 PL=0
MOVL C01149 V=800.0 PL=0
MOVL C01150 V=800.0 PL=0
MOVL C01151 V=800.0 PL=0
MOVL C01152 V=800.0 PL=0
MOVL C01153 V=800.0 PL=0
MOVL C01154 V=800.0 PL=0
MOVL C01155 V=800.0 PL=0
MOVL C01156 V=800.0 PL=0
MOVL C01157 V=800.0 PL=0
MOVL C01158 V=800.0 PL=0
MOVL C01159 V=800.0 PL=0
MOVL C01160 V=800.0 PL=0
MOVL C01161 V=800.0 PL=0
MOVL C01162 V=800.0 PL=0
MOVL C01163 V=800.0 PL=0
MOVL C01164 V=800.0 PL=0
MOVL C01165 V=800.0 PL=0
MOVL C01166 V=800.0 PL=0
MOVL C01167 V=800.0 PL=0
MOVL C01168 V=800.0 PL=0
MOVL C01169 V=800.0 PL=0
MOVL C01170 V=800.0 PL=0
MOVL C01171 V=800.0 PL=0
MOVL C01172 V=800.0 PL=0
MOVL C01173 V=800.0 PL=0
MOVL C01174 V=800.0 PL=0
MOVL C01175 V=800.0 PL=0
MOVL C01176 V=800.0 PL=0
MOVL C01177 V=800.0 PL=0
MOVL C01178 V=800.0 PL=0
MOVL C01179 V=800.0 PL=0
MOVL C01180 V=800.0 PL=0
MOVL C01181 V=800.0 PL=0
MOVL C01182 V=800.0 PL=0
MOVL C01183 V=800.0 PL=0
MOVL C01184 V=800.0 PL=0
MOVL C01185 V=800.0 PL=0
MOVL C01186 V=800.0 PL=0
MOVL C01187 V=800.0 PL=0
MOVL C01188 V=800.0 PL=0
MOVL C01189 V=800.0 PL=0
MOVL C01190 V=800.0 PL=0
MOVL C01191 V=800.0 PL=0
MOVL C01192 V=800.0 PL=0
MOVL C01193 V=800.0 PL=0
MOVL C01194 V=800.0 PL=0
MOVL C01195 V=800.0 PL=0
MOVL C01196 V=800.0 PL=0
MOVL C01197 V=800.0 PL=0
MOVL C01198 V=800.0 PL=0
MOVL C01199 V=800.0 PL=0
MOVL C01200 V=800.0 PL=0
MOVL C01201 V=800.0 PL=0
MOVL C01202 V=800.0 PL=0
MOVL C01203 V=800.0 PL=0
MOVL C01204 V=800.0 PL=0
MOVL C01205 V=800.0 PL=0
MOVL C01206 V=800.0 PL=0
MOVL C01207 V=800.0 PL=0
MOVL C01208 V=800.0 PL=0
MOVL C01209 V=800.0 PL=0
MOVL C01210 V=800.0 PL=0
MOVL C01211 V=800.0 PL=0
MOVL C01212 V=800.0 PL=0
MOVL C01213 V=800.0 PL=0
MOVL C01214 V=800.0 PL=0
MOVL C01215 V=800.0 PL=0
MOVL C01216 V=800.0 PL=0
MOVL C01217 V=800.0 PL=0
MOVL C01218 V=800.0 PL=0
MOVL C01219 V=800.0 PL=0
MOVL C01220 V=800.0 PL=0
MOVL C01221 V=800.0 PL=0
MOVL C01222 V=800.0 PL=0
MOVL C01223 V=800.0 PL=0
MOVL C01224 V=800.0 PL=0
MOVL C01225 V=800.0 PL=0
MOVL C01226 V=800.0 PL=0
MOVL C01227 V=800.0 PL=0
MOVL C01228 V=800.0 PL=0
MOVL C01229 V=800.0 PL=0
MOVL C01230 V=800.0 PL=0
MOVL C01231 V=800.0 PL=0
MOVL C01232 V=800.0 PL=0
MOVL C01233 V=800.0 PL=0
MOVL C01234 V=800.0 PL=0
MOVL C01235 V=800.0 PL=0
MOVL C01236 V=800.0 PL=0
MOVL C01237 V=800.0 PL=0
MOVL C01238 V=800.0 PL=0
MOVL C01239 V=800.0 PL=0
MOVL C01240 V=800.0 PL=0
MOVL C01241 V=800.0 PL=0
MOVL C01242 V=800.0 PL=0
MOVL C01243 V=800.0 PL=0
MOVL C01244 V=800.0 PL=0
MOVL C01245 V=800.0 PL=0
MOVL C01246 V=800.0 PL=0
MOVL C01247 V=800.0 PL=0
MOVL C01248 V=800.0 PL=0
MOVL C01249 V=800.0 PL=0
MOVL C01250 V=800.0 PL=0
MOVL C01251 V=800.0 PL=0
MOVL C01252 V=800.0 PL=0
MOVL C01253 V=800.0 PL=0
MOVL C01254 V=800.0 PL=0
MOVL C01255 V=800.0 PL=0
MOVL C01256 V=800.0 PL=0
MOVL C01257 V=800.0 PL=0
MOVL C01258 V=800.0 PL=0
MOVL C01259 V=800.0 PL=0
MOVL C01260 V=800.0 PL=0
MOVL C01261 V=800.0 PL=0
MOVL C01262 V=800.0 PL=0
MOVL C01263 V=800.0 PL=0
MOVL C01264 V=800.0 PL=0
MOVL C01265 V=800.0 PL=0
MOVL C01266 V=800.0 PL=0
MOVL C01267 V=800.0 PL=0
MOVL C01268 V=800.0 PL=0
MOVL C01269 V=800.0 PL=0
MOVL C01270 V=800.0 PL=0
MOVL C01271 V=800.0 PL=0
MOVL C01272 V=800.0 PL=0
MOVL C01273 V=800.0 PL=0
MOVL C01274 V=800.0 PL=0
MOVL C01275 V=800.0 PL=0
MOVL C01276 V=800.0 PL=0
MOVL C01277 V=800.0 PL=0
MOVL C01278 V=800.0 PL=0
MOVL C01279 V=800.0 PL=0
MOVL C01280 V=800.0 PL=0
MOVL C01281 V=800.0 PL=0
MOVL C01282 V=800.0 PL=0
MOVL C01283 V=800.0 PL=0
MOVL C01284 V=800.0 PL=0
MOVL C01285 V=800.0 PL=0
MOVL C01286 V=800.0 PL=0
MOVL C01287 V=800.0 PL=0
MOVL C01288 V=800.0 PL=0
MOVL C01289 V=800.0 PL=0
MOVL C01290 V=800.0 PL=0
MOVL C01291 V=800.0 PL=0
MOVL C01292 V=800.0 PL=0
MOVL C01293 V=800.0 PL=0
MOVL C01294 V=800.0 PL=0
MOVL C01295 V=800.0 PL=0
MOVL C01296 V=800.0 PL=0
MOVL C01297 V=800.0 PL=0
MOVL C01298 V=800.0 PL=0
MOVL C01299 V=800.0 PL=0
MOVL C01300 V=800.0 PL=0
MOVL C01301 V=800.0 PL=0
MOVL C01302 V=800.0 PL=0
MOVL C01303 V=800.0 PL=0
MOVL C01304 V=800.0 PL=0
MOVL C01305 V=800.0 PL=0
MOVL C01306 V=800.0 PL=0
MOVL C01307 V=800.0 PL=0
MOVL C01308 V=800.0 PL=0
MOVL C01309 V=800.0 PL=0
MOVL C01310 V=800.0 PL=0
MOVL C01311 V=800.0 PL=0
MOVL C01312 V=800.0 PL=0
MOVL C01313 V=800.0 PL=0
MOVL C01314 V=800.0 PL=0
MOVL C01315 V=800.0 PL=0
MOVL C01316 V=800.0 PL=0
MOVL C01317 V=800.0 PL=0
MOVL C01318 V=800.0 PL=0
MOVL C01319 V=800.0 PL=0
MOVL C01320 V=800.0 PL=0
MOVL C01321 V=800.0 PL=0
MOVL C01322 V=800.0 PL=0
MOVL C01323 V=800.0 PL=0
MOVL C01324 V=800.0 PL=0
MOVL C01325 V=800.0 PL=0
MOVL C01326 V=800.0 PL=0
MOVL C01327 V=800.0 PL=0
MOVL C01328 V=800.0 PL=0
MOVL C01329 V=800.0 PL=0
MOVL C01330 V=800.0 PL=0
MOVL C01331 V=800.0 PL=0
MOVL C01332 V=800.0 PL=0
MOVL C01333 V=800.0 PL=0
MOVL C01334 V=800.0 PL=0
MOVL C01335 V=800.0 PL=0
MOVL C01336 V=800.0 PL=0
MOVL C01337 V=800.0 PL=0
MOVL C01338 V=800.0 PL=0
MOVL C01339 V=800.0 PL=0
MOVL C01340 V=800.0 PL=0
MOVL C01341 V=800.0 PL=0
MOVL C01342 V=800.0 PL=0
MOVL C01343 V=800.0 PL=0
MOVL C01344 V=800.0 PL=0
MOVL C01345 V=800.0 PL=0
MOVL C01346 V=800.0 PL=0
MOVL C01347 V=800.0 PL=0
MOVL C01348 V=800.0 PL=0
MOVL C01349 V=800.0 PL=0
MOVL C01350 V=800.0 PL=0
MOVL C01351 V=800.0 PL=0
MOVL C01352 V=800.0 PL=0
MOVL C01353 V=800.0 PL=0
MOVL C01354 V=800.0 PL=0
MOVL C01355 V=800.0 PL=0
MOVL C01356 V=800.0 PL=0
MOVL C01357 V=800.0 PL=0
MOVL C01358 V=800.0 PL=0
MOVL C01359 V=800.0 PL=0
MOVL C01360 V=800.0 PL=0
MOVL C01361 V=800.0 PL=0
MOVL C01362 V=800.0 PL=0
MOVL C01363 V=800.0 PL=0
MOVL C01364 V=800.0 PL=0
MOVL C01365 V=800.0 PL=0
MOVL C01366 V=800.0 PL=0
MOVL C01367 V=800.0 PL=0
MOVL C01368 V=800.0 PL=0
MOVL C01369 V=800.0 PL=0
MOVL C01370 V=800.0 PL=0
MOVL C01371 V=800.0 PL=0
MOVL C01372 V=800.0 PL=0
MOVL C01373 V=800.0 PL=0
MOVL C01374 V=800.0 PL=0
MOVL C01375 V=800.0 PL=0
MOVL C01376 V=800.0 PL=0
MOVL C01377 V=800.0 PL=0
MOVL C01378 V=800.0 PL=0
MOVL C01379 V=800.0 PL=0
MOVL C01380 V=800.0 PL=0
MOVL C01381 V=800.0 PL=0
MOVL C01382 V=800.0 PL=0
MOVL C01383 V=800.0 PL=0
MOVL C01384 V=800.0 PL=0
MOVL C01385 V=800.0 PL=0
MOVL C01386 V=800.0 PL=0
MOVL C01387 V=800.0 PL=0
MOVL C01388 V=800.0 PL=0
MOVL C01389 V=800.0 PL=0
MOVL C01390 V=800.0 PL=0
MOVL C01391 V=800.0 PL=0
MOVL C01392 V=800.0 PL=0
MOVL C01393 V=800.0 PL=0
MOVL C01394 V=800.0 PL=0
MOVL C01395 V=800.0 PL=0
MOVL C01396 V=800.0 PL=0
MOVL C01397 V=800.0 PL=0
MOVL C01398 V=800.0 PL=0
MOVL C01399 V=800.0 PL=0
MOVL C01400 V=800.0 PL=0
MOVL C01401 V=800.0 PL=0
MOVL C01402 V=800.0 PL=0
MOVL C01403 V=800.0 PL=0
MOVL C01404 V=800.0 PL=0
MOVL C01405 V=800.0 PL=0
MOVL C01406 V=800.0 PL=0
MOVL C01407 V=800.0 PL=0
MOVL C01408 V=800.0 PL=0
MOVL C01409 V=800.0 PL=0
MOVL C01410 V=800.0 PL=0
MOVL C01411 V=800.0 PL=0
MOVL C01412 V=800.0 PL=0
MOVL C01413 V=800.0 PL=0
MOVL C01414 V=800.0 PL=0
MOVL C01415 V=800.0 PL=0
MOVL C01416 V=800.0 PL=0
MOVL C01417 V=800.0 PL=0
MOVL C01418 V=800.0 PL=0
MOVL C01419 V=800.0 PL=0
MOVL C01420 V=800.0 PL=0
MOVL C01421 V=800.0 PL=0
MOVL C01422 V=800.0 PL=0
MOVL C01423 V=800.0 PL=0
MOVL C01424 V=800.0 PL=0
MOVL C01425 V=800.0 PL=0
MOVL C01426 V=800.0 PL=0
MOVL C01427 V=800.0 PL=0
MOVL C01428 V=800.0 PL=0
MOVL C01429 V=800.0 PL=0
MOVL C01430 V=800.0 PL=0
MOVL C01431 V=800.0 PL=0
MOVL C01432 V=800.0 PL=0
MOVL C01433 V=800.0 PL=0
MOVL C01434 V=800.0 PL=0
MOVL C01435 V=800.0 PL=0
MOVL C01436 V=800.0 PL=0
MOVL C01437 V=800.0 PL=0
MOVL C01438 V=800.0 PL=0
MOVL C01439 V=800.0 PL=0
MOVL C01440 V=800.0 PL=0
MOVL C01441 V=800.0 PL=0
MOVL C01442 V=800.0 PL=0
MOVL C01443 V=800.0 PL=0
MOVL C01444 V=800.0 PL=0
MOVL C01445 V=800.0 PL=0
MOVL C01446 V=800.0 PL=0
MOVL C01447 V=800.0 PL=0
MOVL C01448 V=800.0 PL=0
MOVL C01449 V=800.0 PL=0
MOVL C01450 V=800.0 PL=0
MOVL C01451 V=800.0 PL=0
MOVL C01452 V=800.0 PL=0
MOVL C01453 V=800.0 PL=0
MOVL C01454 V=800.0 PL=0
MOVL C01455 V=800.0 PL=0
MOVL C01456 V=800.0 PL=0
MOVL C01457 V=800.0 PL=0
MOVL C01458 V=800.0 PL=0
MOVL C01459 V=800.0 PL=0
MOVL C01460 V=800.0 PL=0
MOVL C01461 V=800.0 PL=0
MOVL C01462 V=800.0 PL=0
MOVL C01463 V=800.0 PL=0
MOVL C01464 V=800.0 PL=0
MOVL C01465 V=800.0 PL=0
MOVL C01466 V=800.0 PL=0
MOVL C01467 V=800.0 PL=0
MOVL C01468 V=800.0 PL=0
MOVL C01469 V=800.0 PL=0
MOVL C01470 V=800.0 PL=0
MOVL C01471 V=800.0 PL=0
MOVL C01472 V=800.0 PL=0
MOVL C01473 V=800.0 PL=0
MOVL C01474 V=800.0 PL=0
MOVL C01475 V=800.0 PL=0
MOVL C01476 V=800.0 PL=0
MOVL C01477 V=800.0 PL=0
MOVL C01478 V=800.0 PL=0
MOVL C01479 V=800.0 PL=0
MOVL C01480 V=800.0 PL=0
MOVL C01481 V=800.0 PL=0
MOVL C01482 V=800.0 PL=0
MOVL C01483 V=800.0 PL=0
MOVL C01484 V=800.0 PL=0
MOVL C01485 V=800.0 PL=0
MOVL C01486 V=800.0 PL=0
MOVL C01487 V=800.0 PL=0
MOVL C01488 V=800.0 PL=0
MOVL C01489 V=800.0 PL=0
MOVL C01490 V=800.0 PL=0
MOVL C01491 V=800.0 PL=0
MOVL C01492 V=800.0 PL=0
MOVL C01493 V=800.0 PL=0
MOVL C01494 V=800.0 PL=0
MOVL C01495 V=800.0 PL=0
MOVL C01496 V=800.0 PL=0
MOVL C01497 V=800.0 PL=0
MOVL C01498 V=800.0 PL=0
MOVL C01499 V=800.0 PL=0
MOVL C01500 V=800.0 PL=0
MOVL C01501 V=800.0 PL=0
MOVL C01502 V=800.0 PL=0
MOVL C01503 V=800.0 PL=0
MOVL C01504 V=800.0 PL=0
MOVL C01505 V=800.0 PL=0
MOVL C01506 V=800.0 PL=0
MOVL C01507 V=800.0 PL=0
MOVL C01508 V=800.0 PL=0
MOVL C01509 V=800.0 PL=0
MOVL C01510 V=800.0 PL=0
MOVL C01511 V=800.0 PL=0
MOVL C01512 V=800.0 PL=0
MOVL C01513 V=800.0 PL=0
MOVL C01514 V=800.0 PL=0
MOVL C01515 V=800.0 PL=0
MOVL C01516 V=800.0 PL=0
MOVL C01517 V=800.0 PL=0
MOVL C01518 V=800.0 PL=0
MOVL C01519 V=800.0 PL=0
MOVL C01520 V=800.0 PL=0
MOVL C01521 V=800.0 PL=0
MOVL C01522 V=800.0 PL=0
MOVL C01523 V=800.0 PL=0
MOVL C01524 V=800.0 PL=0
MOVL C01525 V=800.0 PL=0
MOVL C01526 V=800.0 PL=0
MOVL C01527 V=800.0 PL=0
MOVL C01528 V=800.0 PL=0
MOVL C01529 V=800.0 PL=0
MOVL C01530 V=800.0 PL=0
MOVL C01531 V=800.0 PL=0
MOVL C01532 V=800.0 PL=0
MOVL C01533 V=800.0 PL=0
MOVL C01534 V=800.0 PL=0
MOVL C01535 V=800.0 PL=0
MOVL C01536 V=800.0 PL=0
MOVL C01537 V=800.0 PL=0
MOVL C01538 V=800.0 PL=0
MOVL C01539 V=800.0 PL=0
MOVL C01540 V=800.0 PL=0
MOVL C01541 V=800.0 PL=0
MOVL C01542 V=800.0 PL=0
MOVL C01543 V=800.0 PL=0
MOVL C01544 V=800.0 PL=0
MOVL C01545 V=800.0 PL=0
MOVL C01546 V=800.0 PL=0
MOVL C01547 V=800.0 PL=0
MOVL C01548 V=800.0 PL=0
MOVL C01549 V=800.0 PL=0
MOVL C01550 V=800.0 PL=0
MOVL C01551 V=800.0 PL=0
MOVL C01552 V=800.0 PL=0
MOVL C01553 V=800.0 PL=0
MOVL C01554 V=800.0 PL=0
MOVL C01555 V=800.0 PL=0
MOVL C01556 V=800.0 PL=0
MOVL C01557 V=800.0 PL=0
MOVL C01558 V=800.0 PL=0
MOVL C01559 V=800.0 PL=0
MOVL C01560 V=800.0 PL=0
MOVL C01561 V=800.0 PL=0
MOVL C01562 V=800.0 PL=0
MOVL C01563 V=800.0 PL=0
MOVL C01564 V=800.0 PL=0
MOVL C01565 V=800.0 PL=0
MOVL C01566 V=800.0 PL=0
MOVL C01567 V=800.0 PL=0
MOVL C01568 V=800.0 PL=0
MOVL C01569 V=800.0 PL=0
MOVL C01570 V=800.0 PL=0
MOVL C01571 V=800.0 PL=0
MOVL C01572 V=800.0 PL=0
MOVL C01573 V=800.0 PL=0
MOVL C01574 V=800.0 PL=0
MOVL C01575 V=800.0 PL=0
MOVL C01576 V=800.0 PL=0
MOVL C01577 V=800.0 PL=0
MOVL C01578 V=800.0 PL=0
MOVL C01579 V=800.0 PL=0
MOVL C01580 V=800.0 PL=0
MOVL C01581 V=800.0 PL=0
MOVL C01582 V=800.0 PL=0
MOVL C01583 V=800.0 PL=0
MOVL C01584 V=800.0 PL=0
MOVL C01585 V=800.0 PL=0
MOVL C01586 V=800.0 PL=0
MOVL C01587 V=800.0 PL=0
MOVL C01588 V=800.0 PL=0
MOVL C01589 V=800.0 PL=0
MOVL C01590 V=800.0 PL=0
MOVL C01591 V=800.0 PL=0
MOVL C01592 V=800.0 PL=0
MOVL C01593 V=800.0 PL=0
MOVL C01594 V=800.0 PL=0
MOVL C01595 V=800.0 PL=0
MOVL C01596 V=800.0 PL=0
MOVL C01597 V=800.0 PL=0
MOVL C01598 V=800.0 PL=0
MOVL C01599 V=800.0 PL=0
MOVL C01600 V=800.0 PL=0
MOVL C01601 V=800.0 PL=0
MOVL C01602 V=800.0 PL=0
MOVL C01603 V=800.0 PL=0
MOVL C01604 V=800.0 PL=0
MOVL C01605 V=800.0 PL=0
MOVL C01606 V=800.0 PL=0
MOVL C01607 V=800.0 PL=0
MOVL C01608 V=800.0 PL=0
MOVL C01609 V=800.0 PL=0
MOVL C01610 V=800.0 PL=0
MOVL C01611 V=800.0 PL=0
MOVL C01612 V=800.0 PL=0
MOVL C01613 V=800.0 PL=0
MOVL C01614 V=800.0 PL=0
MOVL C01615 V=800.0 PL=0
MOVL C01616 V=800.0 PL=0
MOVL C01617 V=800.0 PL=0
MOVL C01618 V=800.0 PL=0
MOVL C01619 V=800.0 PL=0
MOVL C01620 V=800.0 PL=0
MOVL C01621 V=800.0 PL=0
MOVL C01622 V=800.0 PL=0
MOVL C01623 V=800.0 PL=0
MOVL C01624 V=800.0 PL=0
MOVL C01625 V=800.0 PL=0
MOVL C01626 V=800.0 PL=0
MOVL C01627 V=800.0 PL=0
MOVL C01628 V=800.0 PL=0
MOVL C01629 V=800.0 PL=0
MOVL C01630 V=800.0 PL=0
MOVL C01631 V=800.0 PL=0
MOVL C01632 V=800.0 PL=0
MOVL C01633 V=800.0 PL=0
MOVL C01634 V=800.0 PL=0
MOVL C01635 V=800.0 PL=0
MOVL C01636 V=800.0 PL=0
MOVL C01637 V=800.0 PL=0
MOVL C01638 V=800.0 PL=0
MOVL C01639 V=800.0 PL=0
MOVL C01640 V=800.0 PL=0
MOVL C01641 V=800.0 PL=0
MOVL C01642 V=800.0 PL=0
MOVL C01643 V=800.0 PL=0
MOVL C01644 V=800.0 PL=0
MOVL C01645 V=800.0 PL=0
MOVL C01646 V=800.0 PL=0
MOVL C01647 V=800.0 PL=0
MOVL C01648 V=800.0 PL=0
MOVL C01649 V=800.0 PL=0
MOVL C01650 V=800.0 PL=0
MOVL C01651 V=800.0 PL=0
MOVL C01652 V=800.0 PL=0
MOVL C01653 V=800.0 PL=0
MOVL C01654 V=800.0 PL=0
MOVL C01655 V=800.0 PL=0
MOVL C01656 V=800.0 PL=0
MOVL C01657 V=800.0 PL=0
MOVL C01658 V=800.0 PL=0
MOVL C01659 V=800.0 PL=0
MOVL C01660 V=800.0 PL=0
MOVL C01661 V=800.0 PL=0
MOVL C01662 V=800.0 PL=0
MOVL C01663 V=800.0 PL=0
MOVL C01664 V=800.0 PL=0
MOVL C01665 V=800.0 PL=0
MOVL C01666 V=800.0 PL=0
MOVL C01667 V=800.0 PL=0
MOVL C01668 V=800.0 PL=0
MOVL C01669 V=800.0 PL=0
MOVL C01670 V=800.0 PL=0
MOVL C01671 V=800.0 PL=0
MOVL C01672 V=800.0 PL=0
MOVL C01673 V=800.0 PL=0
MOVL C01674 V=800.0 PL=0
MOVL C01675 V=800.0 PL=0
MOVL C01676 V=800.0 PL=0
MOVL C01677 V=800.0 PL=0
MOVL C01678 V=800.0 PL=0
MOVL C01679 V=800.0 PL=0
MOVL C01680 V=800.0 PL=0
MOVL C01681 V=800.0 PL=0
MOVL C01682 V=800.0 PL=0
MOVL C01683 V=800.0 PL=0
MOVL C01684 V=800.0 PL=0
MOVL C01685 V=800.0 PL=0
MOVL C01686 V=800.0 PL=0
MOVL C01687 V=800.0 PL=0
MOVL C01688 V=800.0 PL=0
MOVL C01689 V=800.0 PL=0
MOVL C01690 V=800.0 PL=0
MOVL C01691 V=800.0 PL=0
MOVL C01692 V=800.0 PL=0
MOVL C01693 V=800.0 PL=0
MOVL C01694 V=800.0 PL=0
MOVL C01695 V=800.0 PL=0
MOVL C01696 V=800.0 PL=0
MOVL C01697 V=800.0 PL=0
MOVL C01698 V=800.0 PL=0
MOVL C01699 V=800.0 PL=0
MOVL C01700 V=800.0 PL=0
MOVL C01701 V=800.0 PL=0
MOVL C01702 V=800.0 PL=0
MOVL C01703 V=800.0 PL=0
MOVL C01704 V=800.0 PL=0
MOVL C01705 V=800.0 PL=0
MOVL C01706 V=800.0 PL=0
MOVL C01707 V=800.0 PL=0
MOVL C01708 V=800.0 PL=0
MOVL C01709 V=800.0 PL=0
MOVL C01710 V=800.0 PL=0
MOVL C01711 V=800.0 PL=0
MOVL C01712 V=800.0 PL=0
MOVL C01713 V=800.0 PL=0
MOVL C01714 V=800.0 PL=0
MOVL C01715 V=800.0 PL=0
MOVL C01716 V=800.0 PL=0
MOVL C01717 V=800.0 PL=0
MOVL C01718 V=800.0 PL=0
MOVL C01719 V=800.0 PL=0
MOVL C01720 V=800.0 PL=0
MOVL C01721 V=800.0 PL=0
MOVL C01722 V=800.0 PL=0
MOVL C01723 V=800.0 PL=0
MOVL C01724 V=800.0 PL=0
MOVL C01725 V=800.0 PL=0
MOVL C01726 V=800.0 PL=0
MOVL C01727 V=800.0 PL=0
MOVL C01728 V=800.0 PL=0
MOVL C01729 V=800.0 PL=0
MOVL C01730 V=800.0 PL=0
MOVL C01731 V=800.0 PL=0
MOVL C01732 V=800.0 PL=0
MOVL C01733 V=800.0 PL=0
MOVL C01734 V=800.0 PL=0
MOVL C01735 V=800.0 PL=0
MOVL C01736 V=800.0 PL=0
MOVL C01737 V=800.0 PL=0
MOVL C01738 V=800.0 PL=0
MOVL C01739 V=800.0 PL=0
MOVL C01740 V=800.0 PL=0
MOVL C01741 V=800.0 PL=0
MOVL C01742 V=800.0 PL=0
MOVL C01743 V=800.0 PL=0
MOVL C01744 V=800.0 PL=0
MOVL C01745 V=800.0 PL=0
MOVL C01746 V=800.0 PL=0
MOVL C01747 V=800.0 PL=0
MOVL C01748 V=800.0 PL=0
MOVL C01749 V=800.0 PL=0
MOVL C01750 V=800.0 PL=0
MOVL C01751 V=800.0 PL=0
MOVL C01752 V=800.0 PL=0
MOVL C01753 V=800.0 PL=0
MOVL C01754 V=800.0 PL=0
MOVL C01755 V=800.0 PL=0
MOVL C01756 V=800.0 PL=0
MOVL C01757 V=800.0 PL=0
MOVL C01758 V=800.0 PL=0
MOVL C01759 V=800.0 PL=0
MOVL C01760 V=800.0 PL=0
MOVL C01761 V=800.0 PL=0
MOVL C01762 V=800.0 PL=0
MOVL C01763 V=800.0 PL=0
MOVL C01764 V=800.0 PL=0
MOVL C01765 V=800.0 PL=0
MOVL C01766 V=800.0 PL=0
MOVL C01767 V=800.0 PL=0
MOVL C01768 V=800.0 PL=0
MOVL C01769 V=800.0 PL=0
MOVL C01770 V=800.0 PL=0
MOVL C01771 V=800.0 PL=0
MOVL C01772 V=800.0 PL=0
MOVL C01773 V=800.0 PL=0
MOVL C01774 V=800.0 PL=0
MOVL C01775 V=800.0 PL=0
MOVL C01776 V=800.0 PL=0
MOVL C01777 V=800.0 PL=0
MOVL C01778 V=800.0 PL=0
MOVL C01779 V=800.0 PL=0
MOVL C01780 V=800.0 PL=0
MOVL C01781 V=800.0 PL=0
MOVL C01782 V=800.0 PL=0
MOVL C01783 V=800.0 PL=0
MOVL C01784 V=800.0 PL=0
MOVL C01785 V=800.0 PL=0
MOVL C01786 V=800.0 PL=0
MOVL C01787 V=800.0 PL=0
MOVL C01788 V=800.0 PL=0
MOVL C01789 V=800.0 PL=0
MOVL C01790 V=800.0 PL=0
MOVL C01791 V=800.0 PL=0
MOVL C01792 V=800.0 PL=0
MOVL C01793 V=800.0 PL=0
MOVL C01794 V=800.0 PL=0
MOVL C01795 V=800.0 PL=0
MOVL C01796 V=800.0 PL=0
MOVL C01797 V=800.0 PL=0
MOVL C01798 V=800.0 PL=0
MOVL C01799 V=800.0 PL=0
MOVL C01800 V=800.0 PL=0
MOVL C01801 V=800.0 PL=0
MOVL C01802 V=800.0 PL=0
MOVL C01803 V=800.0 PL=0
MOVL C01804 V=800.0 PL=0
MOVL C01805 V=800.0 PL=0
MOVL C01806 V=800.0 PL=0
MOVL C01807 V=800.0 PL=0
MOVL C01808 V=800.0 PL=0
MOVL C01809 V=800.0 PL=0
MOVL C01810 V=800.0 PL=0
MOVL C01811 V=800.0 PL=0
MOVL C01812 V=800.0 PL=0
MOVL C01813 V=800.0 PL=0
MOVL C01814 V=800.0 PL=0
MOVL C01815 V=800.0 PL=0
MOVL C01816 V=800.0 PL=0
MOVL C01817 V=800.0 PL=0
MOVL C01818 V=800.0 PL=0
MOVL C01819 V=800.0 PL=0
MOVL C01820 V=800.0 PL=0
MOVL C01821 V=800.0 PL=0
MOVL C01822 V=800.0 PL=0
MOVL C01823 V=800.0 PL=0
MOVL C01824 V=800.0 PL=0
MOVL C01825 V=800.0 PL=0
MOVL C01826 V=800.0 PL=0
MOVL C01827 V=800.0 PL=0
MOVL C01828 V=800.0 PL=0
MOVL C01829 V=800.0 PL=0
MOVL C01830 V=800.0 PL=0
MOVL C01831 V=800.0 PL=0
MOVL C01832 V=800.0 PL=0
MOVL C01833 V=800.0 PL=0
MOVL C01834 V=800.0 PL=0
MOVL C01835 V=800.0 PL=0
MOVL C01836 V=800.0 PL=0
MOVL C01837 V=800.0 PL=0
MOVL C01838 V=800.0 PL=0
MOVL C01839 V=800.0 PL=0
MOVL C01840 V=800.0 PL=0
MOVL C01841 V=800.0 PL=0
MOVL C01842 V=800.0 PL=0
MOVL C01843 V=800.0 PL=0
MOVL C01844 V=800.0 PL=0
MOVL C01845 V=800.0 PL=0
MOVL C01846 V=800.0 PL=0
MOVL C01847 V=800.0 PL=0
MOVL C01848 V=800.0 PL=0
MOVL C01849 V=800.0 PL=0
MOVL C01850 V=800.0 PL=0
MOVL C01851 V=800.0 PL=0
MOVL C01852 V=800.0 PL=0
MOVL C01853 V=800.0 PL=0
MOVL C01854 V=800.0 PL=0
MOVL C01855 V=800.0 PL=0
MOVL C01856 V=800.0 PL=0
MOVL C01857 V=800.0 PL=0
MOVL C01858 V=800.0 PL=0
MOVL C01859 V=800.0 PL=0
MOVL C01860 V=800.0 PL=0
MOVL C01861 V=800.0 PL=0
MOVL C01862 V=800.0 PL=0
MOVL C01863 V=800.0 PL=0
MOVL C01864 V=800.0 PL=0
MOVL C01865 V=800.0 PL=0
MOVL C01866 V=800.0 PL=0
MOVL C01867 V=800.0 PL=0
MOVL C01868 V=800.0 PL=0
MOVL C01869 V=800.0 PL=0
MOVL C01870 V=800.0 PL=0
MOVL C01871 V=800.0 PL=0
MOVL C01872 V=800.0 PL=0
MOVL C01873 V=800.0 PL=0
MOVL C01874 V=800.0 PL=0
MOVL C01875 V=800.0 PL=0
MOVL C01876 V=800.0 PL=0
MOVL C01877 V=800.0 PL=0
MOVL C01878 V=800.0 PL=0
MOVL C01879 V=800.0 PL=0
MOVL C01880 V=800.0 PL=0
MOVL C01881 V=800.0 PL=0
MOVL C01882 V=800.0 PL=0
MOVL C01883 V=800.0 PL=0
MOVL C01884 V=800.0 PL=0
MOVL C01885 V=800.0 PL=0
MOVL C01886 V=800.0 PL=0
MOVL C01887 V=800.0 PL=0
MOVL C01888 V=800.0 PL=0
MOVL C01889 V=800.0 PL=0
MOVL C01890 V=800.0 PL=0
MOVL C01891 V=800.0 PL=0
MOVL C01892 V=800.0 PL=0
MOVL C01893 V=800.0 PL=0
MOVL C01894 V=800.0 PL=0
MOVL C01895 V=800.0 PL=0
MOVL C01896 V=800.0 PL=0
MOVL C01897 V=800.0 PL=0
MOVL C01898 V=800.0 PL=0
MOVL C01899 V=800.0 PL=0
MOVL C01900 V=800.0 PL=0
MOVL C01901 V=800.0 PL=0
MOVL C01902 V=800.0 PL=0
MOVL C01903 V=800.0 PL=0
MOVL C01904 V=800.0 PL=0
MOVL C01905 V=800.0 PL=0
MOVL C01906 V=800.0 PL=0
MOVL C01907 V=800.0 PL=0
MOVL C01908 V=800.0 PL=0
MOVL C01909 V=800.0 PL=0
MOVL C01910 V=800.0 PL=0
MOVL C01911 V=800.0 PL=0
MOVL C01912 V=800.0 PL=0
MOVL C01913 V=800.0 PL=0
MOVL C01914 V=800.0 PL=0
MOVL C01915 V=800.0 PL=0
MOVL C01916 V=800.0 PL=0
MOVL C01917 V=800.0 PL=0
MOVL C01918 V=800.0 PL=0
MOVL C01919 V=800.0 PL=0
MOVL C01920 V=800.0 PL=0
MOVL C01921 V=800.0 PL=0
MOVL C01922 V=800.0 PL=0
MOVL C01923 V=800.0 PL=0
MOVL C01924 V=800.0 PL=0
MOVL C01925 V=800.0 PL=0
MOVL C01926 V=800.0 PL=0
MOVL C01927 V=800.0 PL=0
MOVL C01928 V=800.0 PL=0
MOVL C01929 V=800.0 PL=0
MOVL C01930 V=800.0 PL=0
MOVL C01931 V=800.0 PL=0
MOVL C01932 V=800.0 PL=0
MOVL C01933 V=800.0 PL=0
MOVL C01934 V=800.0 PL=0
MOVL C01935 V=800.0 PL=0
MOVL C01936 V=800.0 PL=0
MOVL C01937 V=800.0 PL=0
MOVL C01938 V=800.0 PL=0
MOVL C01939 V=800.0 PL=0
MOVL C01940 V=800.0 PL=0
MOVL C01941 V=800.0 PL=0
MOVL C01942 V=800.0 PL=0
MOVL C01943 V=800.0 PL=0
MOVL C01944 V=800.0 PL=0
MOVL C01945 V=800.0 PL=0
MOVL C01946 V=800.0 PL=0
MOVL C01947 V=800.0 PL=0
MOVL C01948 V=800.0 PL=0
MOVL C01949 V=800.0 PL=0
MOVL C01950 V=800.0 PL=0
MOVL C01951 V=800.0 PL=0
MOVL C01952 V=800.0 PL=0
MOVL C01953 V=800.0 PL=0
MOVL C01954 V=800.0 PL=0
MOVL C01955 V=800.0 PL=0
MOVL C01956 V=800.0 PL=0
MOVL C01957 V=800.0 PL=0
MOVL C01958 V=800.0 PL=0
MOVL C01959 V=800.0 PL=0
MOVL C01960 V=800.0 PL=0
MOVL C01961 V=800.0 PL=0
MOVL C01962 V=800.0 PL=0
MOVL C01963 V=800.0 PL=0
MOVL C01964 V=800.0 PL=0
MOVL C01965 V=800.0 PL=0
MOVL C01966 V=800.0 PL=0
MOVL C01967 V=800.0 PL=0
MOVL C01968 V=800.0 PL=0
MOVL C01969 V=800.0 PL=0
MOVL C01970 V=800.0 PL=0
MOVL C01971 V=800.0 PL=0
MOVL C01972 V=800.0 PL=0
MOVL C01973 V=800.0 PL=0
MOVL C01974 V=800.0 PL=0
MOVL C01975 V=800.0 PL=0
MOVL C01976 V=800.0 PL=0
MOVL C01977 V=800.0 PL=0
MOVL C01978 V=800.0 PL=0
MOVL C01979 V=800.0 PL=0
MOVL C01980 V=800.0 PL=0
MOVL C01981 V=800.0 PL=0
MOVL C01982 V=800.0 PL=0
MOVL C01983 V=800.0 PL=0
MOVL C01984 V=800.0 PL=0
MOVL C01985 V=800.0 PL=0
MOVL C01986 V=800.0 PL=0
MOVL C01987 V=800.0 PL=0
MOVL C01988 V=800.0 PL=0
MOVL C01989 V=800.0 PL=0
MOVL C01990 V=800.0 PL=0
MOVL C01991 V=800.0 PL=0
MOVL C01992 V=800.0 PL=0
MOVL C01993 V=800.0 PL=0
MOVL C01994 V=800.0 PL=0
MOVL C01995 V=800.0 PL=0
MOVL C01996 V=800.0 PL=0
MOVL C01997 V=800.0 PL=0
MOVL C01998 V=800.0 PL=0
MOVL C01999 V=800.0 PL=0
MOVL C02000 V=800.0 PL=0
MOVL C02001 V=800.0 PL=0
MOVL C02002 V=800.0 PL=0
MOVL C02003 V=800.0 PL=0
MOVL C02004 V=800.0 PL=0
MOVL C02005 V=800.0 PL=0
MOVL C02006 V=800.0 PL=0
MOVL C02007 V=800.0 PL=0
MOVL C02008 V=800.0 PL=0
MOVL C02009 V=800.0 PL=0
MOVL C02010 V=800.0 PL=0
MOVL C02011 V=800.0 PL=0
MOVL C02012 V=800.0 PL=0
MOVL C02013 V=800.0 PL=0
MOVL C02014 V=800.0 PL=0
MOVL C02015 V=800.0 PL=0
MOVL C02016 V=800.0 PL=0
MOVL C02017 V=800.0 PL=0
MOVL C02018 V=800.0 PL=0
MOVL C02019 V=800.0 PL=0
MOVL C02020 V=800.0 PL=0
MOVL C02021 V=800.0 PL=0
MOVL C02022 V=800.0 PL=0
MOVL C02023 V=800.0 PL=0
MOVL C02024 V=800.0 PL=0
MOVL C02025 V=800.0 PL=0
MOVL C02026 V=800.0 PL=0
MOVL C02027 V=800.0 PL=0
MOVL C02028 V=800.0 PL=0
MOVL C02029 V=800.0 PL=0
MOVL C02030 V=800.0 PL=0
MOVL C02031 V=800.0 PL=0
MOVL C02032 V=800.0 PL=0
MOVL C02033 V=800.0 PL=0
MOVL C02034 V=800.0 PL=0
MOVL C02035 V=800.0 PL=0
MOVL C02036 V=800.0 PL=0
MOVL C02037 V=800.0 PL=0
MOVL C02038 V=800.0 PL=0
MOVL C02039 V=800.0 PL=0
MOVL C02040 V=800.0 PL=0
MOVL C02041 V=800.0 PL=0
MOVL C02042 V=800.0 PL=0
MOVL C02043 V=800.0 PL=0
MOVL C02044 V=800.0 PL=0
MOVL C02045 V=800.0 PL=0
MOVL C02046 V=800.0 PL=0
MOVL C02047 V=800.0 PL=0
MOVL C02048 V=800.0 PL=0
MOVL C02049 V=800.0 PL=0
MOVL C02050 V=800.0 PL=0
MOVL C02051 V=800.0 PL=0
MOVL C02052 V=800.0 PL=0
MOVL C02053 V=800.0 PL=0
MOVL C02054 V=800.0 PL=0
MOVL C02055 V=800.0 PL=0
MOVL C02056 V=800.0 PL=0
MOVL C02057 V=800.0 PL=0
MOVL C02058 V=800.0 PL=0
MOVL C02059 V=800.0 PL=0
MOVL C02060 V=800.0 PL=0
MOVL C02061 V=800.0 PL=0
MOVL C02062 V=800.0 PL=0
MOVL C02063 V=800.0 PL=0
MOVL C02064 V=800.0 PL=0
MOVL C02065 V=800.0 PL=0
MOVL C02066 V=800.0 PL=0
MOVL C02067 V=800.0 PL=0
MOVL C02068 V=800.0 PL=0
MOVL C02069 V=800.0 PL=0
MOVL C02070 V=800.0 PL=0
MOVL C02071 V=800.0 PL=0
MOVL C02072 V=800.0 PL=0
MOVL C02073 V=800.0 PL=0
MOVL C02074 V=800.0 PL=0
MOVL C02075 V=800.0 PL=0
MOVL C02076 V=800.0 PL=0
MOVL C02077 V=800.0 PL=0
MOVL C02078 V=800.0 PL=0
MOVL C02079 V=800.0 PL=0
MOVL C02080 V=800.0 PL=0
MOVL C02081 V=800.0 PL=0
MOVL C02082 V=800.0 PL=0
MOVL C02083 V=800.0 PL=0
MOVL C02084 V=800.0 PL=0
MOVL C02085 V=800.0 PL=0
MOVL C02086 V=800.0 PL=0
MOVL C02087 V=800.0 PL=0
MOVL C02088 V=800.0 PL=0
MOVL C02089 V=800.0 PL=0
MOVL C02090 V=800.0 PL=0
MOVL C02091 V=800.0 PL=0
MOVL C02092 V=800.0 PL=0
MOVL C02093 V=800.0 PL=0
MOVL C02094 V=800.0 PL=0
MOVL C02095 V=800.0 PL=0
MOVL C02096 V=800.0 PL=0
MOVL C02097 V=800.0 PL=0
MOVL C02098 V=800.0 PL=0
MOVL C02099 V=800.0 PL=0
MOVL C02100 V=800.0 PL=0
MOVL C02101 V=800.0 PL=0
MOVL C02102 V=800.0 PL=0
MOVL C02103 V=800.0 PL=0
MOVL C02104 V=800.0 PL=0
MOVL C02105 V=800.0 PL=0
MOVL C02106 V=800.0 PL=0
MOVL C02107 V=800.0 PL=0
MOVL C02108 V=800.0 PL=0
